;FOLD LIN P2461 Vel=2 m/s CPDAT2461 Tool[1]:marker Base[0] ;%{PE}
;FOLD Parameters ;%{h}
;Params IlfProvider=kukaroboter.basistech.inlineforms.movement.old; Kuka.IsGlobalPoint=False; Kuka.PointName=P2461; Kuka.BlendingEnabled=False; Kuka.MoveDataName=CPDAT1; Kuka.VelocityPath=2; Kuka.CurrentCDSetIndex=0; Kuka.MovementParameterFieldEnabled=True; IlfCommand=LIN
;ENDFOLD
$BWDSTART = FALSE
LDAT_ACT = LCPDAT2461
FDAT_ACT = FP2461
BAS(#CP_PARAMS, 2.0)
SET_CD_PARAMS (0)
LIN XP2461
;ENDFOLD

;FOLD LIN P2462 Vel=2 m/s CPDAT2462 Tool[1]:marker Base[0] ;%{PE}
;FOLD Parameters ;%{h}
;Params IlfProvider=kukaroboter.basistech.inlineforms.movement.old; Kuka.IsGlobalPoint=False; Kuka.PointName=P2462; Kuka.BlendingEnabled=False; Kuka.MoveDataName=CPDAT1; Kuka.VelocityPath=2; Kuka.CurrentCDSetIndex=0; Kuka.MovementParameterFieldEnabled=True; IlfCommand=LIN
;ENDFOLD
$BWDSTART = FALSE
LDAT_ACT = LCPDAT2462
FDAT_ACT = FP2462
BAS(#CP_PARAMS, 2.0)
SET_CD_PARAMS (0)
LIN XP2462
;ENDFOLD

;FOLD LIN P2463 Vel=2 m/s CPDAT2463 Tool[1]:marker Base[0] ;%{PE}
;FOLD Parameters ;%{h}
;Params IlfProvider=kukaroboter.basistech.inlineforms.movement.old; Kuka.IsGlobalPoint=False; Kuka.PointName=P2463; Kuka.BlendingEnabled=False; Kuka.MoveDataName=CPDAT1; Kuka.VelocityPath=2; Kuka.CurrentCDSetIndex=0; Kuka.MovementParameterFieldEnabled=True; IlfCommand=LIN
;ENDFOLD
$BWDSTART = FALSE
LDAT_ACT = LCPDAT2463
FDAT_ACT = FP2463
BAS(#CP_PARAMS, 2.0)
SET_CD_PARAMS (0)
LIN XP2463
;ENDFOLD

;FOLD LIN P2464 Vel=2 m/s CPDAT2464 Tool[1]:marker Base[0] ;%{PE}
;FOLD Parameters ;%{h}
;Params IlfProvider=kukaroboter.basistech.inlineforms.movement.old; Kuka.IsGlobalPoint=False; Kuka.PointName=P2464; Kuka.BlendingEnabled=False; Kuka.MoveDataName=CPDAT1; Kuka.VelocityPath=2; Kuka.CurrentCDSetIndex=0; Kuka.MovementParameterFieldEnabled=True; IlfCommand=LIN
;ENDFOLD
$BWDSTART = FALSE
LDAT_ACT = LCPDAT2464
FDAT_ACT = FP2464
BAS(#CP_PARAMS, 2.0)
SET_CD_PARAMS (0)
LIN XP2464
;ENDFOLD

;FOLD LIN P2465 Vel=2 m/s CPDAT2465 Tool[1]:marker Base[0] ;%{PE}
;FOLD Parameters ;%{h}
;Params IlfProvider=kukaroboter.basistech.inlineforms.movement.old; Kuka.IsGlobalPoint=False; Kuka.PointName=P2465; Kuka.BlendingEnabled=False; Kuka.MoveDataName=CPDAT1; Kuka.VelocityPath=2; Kuka.CurrentCDSetIndex=0; Kuka.MovementParameterFieldEnabled=True; IlfCommand=LIN
;ENDFOLD
$BWDSTART = FALSE
LDAT_ACT = LCPDAT2465
FDAT_ACT = FP2465
BAS(#CP_PARAMS, 2.0)
SET_CD_PARAMS (0)
LIN XP2465
;ENDFOLD

;FOLD LIN P2466 Vel=2 m/s CPDAT2466 Tool[1]:marker Base[0] ;%{PE}
;FOLD Parameters ;%{h}
;Params IlfProvider=kukaroboter.basistech.inlineforms.movement.old; Kuka.IsGlobalPoint=False; Kuka.PointName=P2466; Kuka.BlendingEnabled=False; Kuka.MoveDataName=CPDAT1; Kuka.VelocityPath=2; Kuka.CurrentCDSetIndex=0; Kuka.MovementParameterFieldEnabled=True; IlfCommand=LIN
;ENDFOLD
$BWDSTART = FALSE
LDAT_ACT = LCPDAT2466
FDAT_ACT = FP2466
BAS(#CP_PARAMS, 2.0)
SET_CD_PARAMS (0)
LIN XP2466
;ENDFOLD

;FOLD LIN P2467 Vel=2 m/s CPDAT2467 Tool[1]:marker Base[0] ;%{PE}
;FOLD Parameters ;%{h}
;Params IlfProvider=kukaroboter.basistech.inlineforms.movement.old; Kuka.IsGlobalPoint=False; Kuka.PointName=P2467; Kuka.BlendingEnabled=False; Kuka.MoveDataName=CPDAT1; Kuka.VelocityPath=2; Kuka.CurrentCDSetIndex=0; Kuka.MovementParameterFieldEnabled=True; IlfCommand=LIN
;ENDFOLD
$BWDSTART = FALSE
LDAT_ACT = LCPDAT2467
FDAT_ACT = FP2467
BAS(#CP_PARAMS, 2.0)
SET_CD_PARAMS (0)
LIN XP2467
;ENDFOLD

;FOLD LIN P2468 Vel=2 m/s CPDAT2468 Tool[1]:marker Base[0] ;%{PE}
;FOLD Parameters ;%{h}
;Params IlfProvider=kukaroboter.basistech.inlineforms.movement.old; Kuka.IsGlobalPoint=False; Kuka.PointName=P2468; Kuka.BlendingEnabled=False; Kuka.MoveDataName=CPDAT1; Kuka.VelocityPath=2; Kuka.CurrentCDSetIndex=0; Kuka.MovementParameterFieldEnabled=True; IlfCommand=LIN
;ENDFOLD
$BWDSTART = FALSE
LDAT_ACT = LCPDAT2468
FDAT_ACT = FP2468
BAS(#CP_PARAMS, 2.0)
SET_CD_PARAMS (0)
LIN XP2468
;ENDFOLD

;FOLD LIN P2469 Vel=2 m/s CPDAT2469 Tool[1]:marker Base[0] ;%{PE}
;FOLD Parameters ;%{h}
;Params IlfProvider=kukaroboter.basistech.inlineforms.movement.old; Kuka.IsGlobalPoint=False; Kuka.PointName=P2469; Kuka.BlendingEnabled=False; Kuka.MoveDataName=CPDAT1; Kuka.VelocityPath=2; Kuka.CurrentCDSetIndex=0; Kuka.MovementParameterFieldEnabled=True; IlfCommand=LIN
;ENDFOLD
$BWDSTART = FALSE
LDAT_ACT = LCPDAT2469
FDAT_ACT = FP2469
BAS(#CP_PARAMS, 2.0)
SET_CD_PARAMS (0)
LIN XP2469
;ENDFOLD

;FOLD LIN P2470 Vel=2 m/s CPDAT2470 Tool[1]:marker Base[0] ;%{PE}
;FOLD Parameters ;%{h}
;Params IlfProvider=kukaroboter.basistech.inlineforms.movement.old; Kuka.IsGlobalPoint=False; Kuka.PointName=P2470; Kuka.BlendingEnabled=False; Kuka.MoveDataName=CPDAT1; Kuka.VelocityPath=2; Kuka.CurrentCDSetIndex=0; Kuka.MovementParameterFieldEnabled=True; IlfCommand=LIN
;ENDFOLD
$BWDSTART = FALSE
LDAT_ACT = LCPDAT2470
FDAT_ACT = FP2470
BAS(#CP_PARAMS, 2.0)
SET_CD_PARAMS (0)
LIN XP2470
;ENDFOLD

;FOLD LIN P2471 Vel=2 m/s CPDAT2471 Tool[1]:marker Base[0] ;%{PE}
;FOLD Parameters ;%{h}
;Params IlfProvider=kukaroboter.basistech.inlineforms.movement.old; Kuka.IsGlobalPoint=False; Kuka.PointName=P2471; Kuka.BlendingEnabled=False; Kuka.MoveDataName=CPDAT1; Kuka.VelocityPath=2; Kuka.CurrentCDSetIndex=0; Kuka.MovementParameterFieldEnabled=True; IlfCommand=LIN
;ENDFOLD
$BWDSTART = FALSE
LDAT_ACT = LCPDAT2471
FDAT_ACT = FP2471
BAS(#CP_PARAMS, 2.0)
SET_CD_PARAMS (0)
LIN XP2471
;ENDFOLD

;FOLD LIN P2472 Vel=2 m/s CPDAT2472 Tool[1]:marker Base[0] ;%{PE}
;FOLD Parameters ;%{h}
;Params IlfProvider=kukaroboter.basistech.inlineforms.movement.old; Kuka.IsGlobalPoint=False; Kuka.PointName=P2472; Kuka.BlendingEnabled=False; Kuka.MoveDataName=CPDAT1; Kuka.VelocityPath=2; Kuka.CurrentCDSetIndex=0; Kuka.MovementParameterFieldEnabled=True; IlfCommand=LIN
;ENDFOLD
$BWDSTART = FALSE
LDAT_ACT = LCPDAT2472
FDAT_ACT = FP2472
BAS(#CP_PARAMS, 2.0)
SET_CD_PARAMS (0)
LIN XP2472
;ENDFOLD

;FOLD LIN P2473 Vel=2 m/s CPDAT2473 Tool[1]:marker Base[0] ;%{PE}
;FOLD Parameters ;%{h}
;Params IlfProvider=kukaroboter.basistech.inlineforms.movement.old; Kuka.IsGlobalPoint=False; Kuka.PointName=P2473; Kuka.BlendingEnabled=False; Kuka.MoveDataName=CPDAT1; Kuka.VelocityPath=2; Kuka.CurrentCDSetIndex=0; Kuka.MovementParameterFieldEnabled=True; IlfCommand=LIN
;ENDFOLD
$BWDSTART = FALSE
LDAT_ACT = LCPDAT2473
FDAT_ACT = FP2473
BAS(#CP_PARAMS, 2.0)
SET_CD_PARAMS (0)
LIN XP2473
;ENDFOLD

;FOLD LIN P2474 Vel=2 m/s CPDAT2474 Tool[1]:marker Base[0] ;%{PE}
;FOLD Parameters ;%{h}
;Params IlfProvider=kukaroboter.basistech.inlineforms.movement.old; Kuka.IsGlobalPoint=False; Kuka.PointName=P2474; Kuka.BlendingEnabled=False; Kuka.MoveDataName=CPDAT1; Kuka.VelocityPath=2; Kuka.CurrentCDSetIndex=0; Kuka.MovementParameterFieldEnabled=True; IlfCommand=LIN
;ENDFOLD
$BWDSTART = FALSE
LDAT_ACT = LCPDAT2474
FDAT_ACT = FP2474
BAS(#CP_PARAMS, 2.0)
SET_CD_PARAMS (0)
LIN XP2474
;ENDFOLD

;FOLD LIN P2475 Vel=2 m/s CPDAT2475 Tool[1]:marker Base[0] ;%{PE}
;FOLD Parameters ;%{h}
;Params IlfProvider=kukaroboter.basistech.inlineforms.movement.old; Kuka.IsGlobalPoint=False; Kuka.PointName=P2475; Kuka.BlendingEnabled=False; Kuka.MoveDataName=CPDAT1; Kuka.VelocityPath=2; Kuka.CurrentCDSetIndex=0; Kuka.MovementParameterFieldEnabled=True; IlfCommand=LIN
;ENDFOLD
$BWDSTART = FALSE
LDAT_ACT = LCPDAT2475
FDAT_ACT = FP2475
BAS(#CP_PARAMS, 2.0)
SET_CD_PARAMS (0)
LIN XP2475
;ENDFOLD

;FOLD LIN P2476 Vel=2 m/s CPDAT2476 Tool[1]:marker Base[0] ;%{PE}
;FOLD Parameters ;%{h}
;Params IlfProvider=kukaroboter.basistech.inlineforms.movement.old; Kuka.IsGlobalPoint=False; Kuka.PointName=P2476; Kuka.BlendingEnabled=False; Kuka.MoveDataName=CPDAT1; Kuka.VelocityPath=2; Kuka.CurrentCDSetIndex=0; Kuka.MovementParameterFieldEnabled=True; IlfCommand=LIN
;ENDFOLD
$BWDSTART = FALSE
LDAT_ACT = LCPDAT2476
FDAT_ACT = FP2476
BAS(#CP_PARAMS, 2.0)
SET_CD_PARAMS (0)
LIN XP2476
;ENDFOLD

;FOLD LIN P2477 Vel=2 m/s CPDAT2477 Tool[1]:marker Base[0] ;%{PE}
;FOLD Parameters ;%{h}
;Params IlfProvider=kukaroboter.basistech.inlineforms.movement.old; Kuka.IsGlobalPoint=False; Kuka.PointName=P2477; Kuka.BlendingEnabled=False; Kuka.MoveDataName=CPDAT1; Kuka.VelocityPath=2; Kuka.CurrentCDSetIndex=0; Kuka.MovementParameterFieldEnabled=True; IlfCommand=LIN
;ENDFOLD
$BWDSTART = FALSE
LDAT_ACT = LCPDAT2477
FDAT_ACT = FP2477
BAS(#CP_PARAMS, 2.0)
SET_CD_PARAMS (0)
LIN XP2477
;ENDFOLD

;FOLD LIN P2478 Vel=2 m/s CPDAT2478 Tool[1]:marker Base[0] ;%{PE}
;FOLD Parameters ;%{h}
;Params IlfProvider=kukaroboter.basistech.inlineforms.movement.old; Kuka.IsGlobalPoint=False; Kuka.PointName=P2478; Kuka.BlendingEnabled=False; Kuka.MoveDataName=CPDAT1; Kuka.VelocityPath=2; Kuka.CurrentCDSetIndex=0; Kuka.MovementParameterFieldEnabled=True; IlfCommand=LIN
;ENDFOLD
$BWDSTART = FALSE
LDAT_ACT = LCPDAT2478
FDAT_ACT = FP2478
BAS(#CP_PARAMS, 2.0)
SET_CD_PARAMS (0)
LIN XP2478
;ENDFOLD

;FOLD LIN P2479 Vel=2 m/s CPDAT2479 Tool[1]:marker Base[0] ;%{PE}
;FOLD Parameters ;%{h}
;Params IlfProvider=kukaroboter.basistech.inlineforms.movement.old; Kuka.IsGlobalPoint=False; Kuka.PointName=P2479; Kuka.BlendingEnabled=False; Kuka.MoveDataName=CPDAT1; Kuka.VelocityPath=2; Kuka.CurrentCDSetIndex=0; Kuka.MovementParameterFieldEnabled=True; IlfCommand=LIN
;ENDFOLD
$BWDSTART = FALSE
LDAT_ACT = LCPDAT2479
FDAT_ACT = FP2479
BAS(#CP_PARAMS, 2.0)
SET_CD_PARAMS (0)
LIN XP2479
;ENDFOLD

;FOLD LIN P2480 Vel=2 m/s CPDAT2480 Tool[1]:marker Base[0] ;%{PE}
;FOLD Parameters ;%{h}
;Params IlfProvider=kukaroboter.basistech.inlineforms.movement.old; Kuka.IsGlobalPoint=False; Kuka.PointName=P2480; Kuka.BlendingEnabled=False; Kuka.MoveDataName=CPDAT1; Kuka.VelocityPath=2; Kuka.CurrentCDSetIndex=0; Kuka.MovementParameterFieldEnabled=True; IlfCommand=LIN
;ENDFOLD
$BWDSTART = FALSE
LDAT_ACT = LCPDAT2480
FDAT_ACT = FP2480
BAS(#CP_PARAMS, 2.0)
SET_CD_PARAMS (0)
LIN XP2480
;ENDFOLD

;FOLD LIN P2481 Vel=2 m/s CPDAT2481 Tool[1]:marker Base[0] ;%{PE}
;FOLD Parameters ;%{h}
;Params IlfProvider=kukaroboter.basistech.inlineforms.movement.old; Kuka.IsGlobalPoint=False; Kuka.PointName=P2481; Kuka.BlendingEnabled=False; Kuka.MoveDataName=CPDAT1; Kuka.VelocityPath=2; Kuka.CurrentCDSetIndex=0; Kuka.MovementParameterFieldEnabled=True; IlfCommand=LIN
;ENDFOLD
$BWDSTART = FALSE
LDAT_ACT = LCPDAT2481
FDAT_ACT = FP2481
BAS(#CP_PARAMS, 2.0)
SET_CD_PARAMS (0)
LIN XP2481
;ENDFOLD

;FOLD LIN P2482 Vel=2 m/s CPDAT2482 Tool[1]:marker Base[0] ;%{PE}
;FOLD Parameters ;%{h}
;Params IlfProvider=kukaroboter.basistech.inlineforms.movement.old; Kuka.IsGlobalPoint=False; Kuka.PointName=P2482; Kuka.BlendingEnabled=False; Kuka.MoveDataName=CPDAT1; Kuka.VelocityPath=2; Kuka.CurrentCDSetIndex=0; Kuka.MovementParameterFieldEnabled=True; IlfCommand=LIN
;ENDFOLD
$BWDSTART = FALSE
LDAT_ACT = LCPDAT2482
FDAT_ACT = FP2482
BAS(#CP_PARAMS, 2.0)
SET_CD_PARAMS (0)
LIN XP2482
;ENDFOLD

;FOLD LIN P2483 Vel=2 m/s CPDAT2483 Tool[1]:marker Base[0] ;%{PE}
;FOLD Parameters ;%{h}
;Params IlfProvider=kukaroboter.basistech.inlineforms.movement.old; Kuka.IsGlobalPoint=False; Kuka.PointName=P2483; Kuka.BlendingEnabled=False; Kuka.MoveDataName=CPDAT1; Kuka.VelocityPath=2; Kuka.CurrentCDSetIndex=0; Kuka.MovementParameterFieldEnabled=True; IlfCommand=LIN
;ENDFOLD
$BWDSTART = FALSE
LDAT_ACT = LCPDAT2483
FDAT_ACT = FP2483
BAS(#CP_PARAMS, 2.0)
SET_CD_PARAMS (0)
LIN XP2483
;ENDFOLD

;FOLD LIN P2484 Vel=2 m/s CPDAT2484 Tool[1]:marker Base[0] ;%{PE}
;FOLD Parameters ;%{h}
;Params IlfProvider=kukaroboter.basistech.inlineforms.movement.old; Kuka.IsGlobalPoint=False; Kuka.PointName=P2484; Kuka.BlendingEnabled=False; Kuka.MoveDataName=CPDAT1; Kuka.VelocityPath=2; Kuka.CurrentCDSetIndex=0; Kuka.MovementParameterFieldEnabled=True; IlfCommand=LIN
;ENDFOLD
$BWDSTART = FALSE
LDAT_ACT = LCPDAT2484
FDAT_ACT = FP2484
BAS(#CP_PARAMS, 2.0)
SET_CD_PARAMS (0)
LIN XP2484
;ENDFOLD

;FOLD LIN P2485 Vel=2 m/s CPDAT2485 Tool[1]:marker Base[0] ;%{PE}
;FOLD Parameters ;%{h}
;Params IlfProvider=kukaroboter.basistech.inlineforms.movement.old; Kuka.IsGlobalPoint=False; Kuka.PointName=P2485; Kuka.BlendingEnabled=False; Kuka.MoveDataName=CPDAT1; Kuka.VelocityPath=2; Kuka.CurrentCDSetIndex=0; Kuka.MovementParameterFieldEnabled=True; IlfCommand=LIN
;ENDFOLD
$BWDSTART = FALSE
LDAT_ACT = LCPDAT2485
FDAT_ACT = FP2485
BAS(#CP_PARAMS, 2.0)
SET_CD_PARAMS (0)
LIN XP2485
;ENDFOLD

;FOLD LIN P2486 Vel=2 m/s CPDAT2486 Tool[1]:marker Base[0] ;%{PE}
;FOLD Parameters ;%{h}
;Params IlfProvider=kukaroboter.basistech.inlineforms.movement.old; Kuka.IsGlobalPoint=False; Kuka.PointName=P2486; Kuka.BlendingEnabled=False; Kuka.MoveDataName=CPDAT1; Kuka.VelocityPath=2; Kuka.CurrentCDSetIndex=0; Kuka.MovementParameterFieldEnabled=True; IlfCommand=LIN
;ENDFOLD
$BWDSTART = FALSE
LDAT_ACT = LCPDAT2486
FDAT_ACT = FP2486
BAS(#CP_PARAMS, 2.0)
SET_CD_PARAMS (0)
LIN XP2486
;ENDFOLD

;FOLD LIN P2487 Vel=2 m/s CPDAT2487 Tool[1]:marker Base[0] ;%{PE}
;FOLD Parameters ;%{h}
;Params IlfProvider=kukaroboter.basistech.inlineforms.movement.old; Kuka.IsGlobalPoint=False; Kuka.PointName=P2487; Kuka.BlendingEnabled=False; Kuka.MoveDataName=CPDAT1; Kuka.VelocityPath=2; Kuka.CurrentCDSetIndex=0; Kuka.MovementParameterFieldEnabled=True; IlfCommand=LIN
;ENDFOLD
$BWDSTART = FALSE
LDAT_ACT = LCPDAT2487
FDAT_ACT = FP2487
BAS(#CP_PARAMS, 2.0)
SET_CD_PARAMS (0)
LIN XP2487
;ENDFOLD

;FOLD LIN P2488 Vel=2 m/s CPDAT2488 Tool[1]:marker Base[0] ;%{PE}
;FOLD Parameters ;%{h}
;Params IlfProvider=kukaroboter.basistech.inlineforms.movement.old; Kuka.IsGlobalPoint=False; Kuka.PointName=P2488; Kuka.BlendingEnabled=False; Kuka.MoveDataName=CPDAT1; Kuka.VelocityPath=2; Kuka.CurrentCDSetIndex=0; Kuka.MovementParameterFieldEnabled=True; IlfCommand=LIN
;ENDFOLD
$BWDSTART = FALSE
LDAT_ACT = LCPDAT2488
FDAT_ACT = FP2488
BAS(#CP_PARAMS, 2.0)
SET_CD_PARAMS (0)
LIN XP2488
;ENDFOLD

;FOLD LIN P2489 Vel=2 m/s CPDAT2489 Tool[1]:marker Base[0] ;%{PE}
;FOLD Parameters ;%{h}
;Params IlfProvider=kukaroboter.basistech.inlineforms.movement.old; Kuka.IsGlobalPoint=False; Kuka.PointName=P2489; Kuka.BlendingEnabled=False; Kuka.MoveDataName=CPDAT1; Kuka.VelocityPath=2; Kuka.CurrentCDSetIndex=0; Kuka.MovementParameterFieldEnabled=True; IlfCommand=LIN
;ENDFOLD
$BWDSTART = FALSE
LDAT_ACT = LCPDAT2489
FDAT_ACT = FP2489
BAS(#CP_PARAMS, 2.0)
SET_CD_PARAMS (0)
LIN XP2489
;ENDFOLD

;FOLD LIN P2490 Vel=2 m/s CPDAT2490 Tool[1]:marker Base[0] ;%{PE}
;FOLD Parameters ;%{h}
;Params IlfProvider=kukaroboter.basistech.inlineforms.movement.old; Kuka.IsGlobalPoint=False; Kuka.PointName=P2490; Kuka.BlendingEnabled=False; Kuka.MoveDataName=CPDAT1; Kuka.VelocityPath=2; Kuka.CurrentCDSetIndex=0; Kuka.MovementParameterFieldEnabled=True; IlfCommand=LIN
;ENDFOLD
$BWDSTART = FALSE
LDAT_ACT = LCPDAT2490
FDAT_ACT = FP2490
BAS(#CP_PARAMS, 2.0)
SET_CD_PARAMS (0)
LIN XP2490
;ENDFOLD

;FOLD LIN P2491 Vel=2 m/s CPDAT2491 Tool[1]:marker Base[0] ;%{PE}
;FOLD Parameters ;%{h}
;Params IlfProvider=kukaroboter.basistech.inlineforms.movement.old; Kuka.IsGlobalPoint=False; Kuka.PointName=P2491; Kuka.BlendingEnabled=False; Kuka.MoveDataName=CPDAT1; Kuka.VelocityPath=2; Kuka.CurrentCDSetIndex=0; Kuka.MovementParameterFieldEnabled=True; IlfCommand=LIN
;ENDFOLD
$BWDSTART = FALSE
LDAT_ACT = LCPDAT2491
FDAT_ACT = FP2491
BAS(#CP_PARAMS, 2.0)
SET_CD_PARAMS (0)
LIN XP2491
;ENDFOLD

;FOLD LIN P2492 Vel=2 m/s CPDAT2492 Tool[1]:marker Base[0] ;%{PE}
;FOLD Parameters ;%{h}
;Params IlfProvider=kukaroboter.basistech.inlineforms.movement.old; Kuka.IsGlobalPoint=False; Kuka.PointName=P2492; Kuka.BlendingEnabled=False; Kuka.MoveDataName=CPDAT1; Kuka.VelocityPath=2; Kuka.CurrentCDSetIndex=0; Kuka.MovementParameterFieldEnabled=True; IlfCommand=LIN
;ENDFOLD
$BWDSTART = FALSE
LDAT_ACT = LCPDAT2492
FDAT_ACT = FP2492
BAS(#CP_PARAMS, 2.0)
SET_CD_PARAMS (0)
LIN XP2492
;ENDFOLD

;FOLD LIN P2493 Vel=2 m/s CPDAT2493 Tool[1]:marker Base[0] ;%{PE}
;FOLD Parameters ;%{h}
;Params IlfProvider=kukaroboter.basistech.inlineforms.movement.old; Kuka.IsGlobalPoint=False; Kuka.PointName=P2493; Kuka.BlendingEnabled=False; Kuka.MoveDataName=CPDAT1; Kuka.VelocityPath=2; Kuka.CurrentCDSetIndex=0; Kuka.MovementParameterFieldEnabled=True; IlfCommand=LIN
;ENDFOLD
$BWDSTART = FALSE
LDAT_ACT = LCPDAT2493
FDAT_ACT = FP2493
BAS(#CP_PARAMS, 2.0)
SET_CD_PARAMS (0)
LIN XP2493
;ENDFOLD

;FOLD LIN P2494 Vel=2 m/s CPDAT2494 Tool[1]:marker Base[0] ;%{PE}
;FOLD Parameters ;%{h}
;Params IlfProvider=kukaroboter.basistech.inlineforms.movement.old; Kuka.IsGlobalPoint=False; Kuka.PointName=P2494; Kuka.BlendingEnabled=False; Kuka.MoveDataName=CPDAT1; Kuka.VelocityPath=2; Kuka.CurrentCDSetIndex=0; Kuka.MovementParameterFieldEnabled=True; IlfCommand=LIN
;ENDFOLD
$BWDSTART = FALSE
LDAT_ACT = LCPDAT2494
FDAT_ACT = FP2494
BAS(#CP_PARAMS, 2.0)
SET_CD_PARAMS (0)
LIN XP2494
;ENDFOLD

;FOLD LIN P2495 Vel=2 m/s CPDAT2495 Tool[1]:marker Base[0] ;%{PE}
;FOLD Parameters ;%{h}
;Params IlfProvider=kukaroboter.basistech.inlineforms.movement.old; Kuka.IsGlobalPoint=False; Kuka.PointName=P2495; Kuka.BlendingEnabled=False; Kuka.MoveDataName=CPDAT1; Kuka.VelocityPath=2; Kuka.CurrentCDSetIndex=0; Kuka.MovementParameterFieldEnabled=True; IlfCommand=LIN
;ENDFOLD
$BWDSTART = FALSE
LDAT_ACT = LCPDAT2495
FDAT_ACT = FP2495
BAS(#CP_PARAMS, 2.0)
SET_CD_PARAMS (0)
LIN XP2495
;ENDFOLD

;FOLD LIN P2496 Vel=2 m/s CPDAT2496 Tool[1]:marker Base[0] ;%{PE}
;FOLD Parameters ;%{h}
;Params IlfProvider=kukaroboter.basistech.inlineforms.movement.old; Kuka.IsGlobalPoint=False; Kuka.PointName=P2496; Kuka.BlendingEnabled=False; Kuka.MoveDataName=CPDAT1; Kuka.VelocityPath=2; Kuka.CurrentCDSetIndex=0; Kuka.MovementParameterFieldEnabled=True; IlfCommand=LIN
;ENDFOLD
$BWDSTART = FALSE
LDAT_ACT = LCPDAT2496
FDAT_ACT = FP2496
BAS(#CP_PARAMS, 2.0)
SET_CD_PARAMS (0)
LIN XP2496
;ENDFOLD

;FOLD LIN P2497 Vel=2 m/s CPDAT2497 Tool[1]:marker Base[0] ;%{PE}
;FOLD Parameters ;%{h}
;Params IlfProvider=kukaroboter.basistech.inlineforms.movement.old; Kuka.IsGlobalPoint=False; Kuka.PointName=P2497; Kuka.BlendingEnabled=False; Kuka.MoveDataName=CPDAT1; Kuka.VelocityPath=2; Kuka.CurrentCDSetIndex=0; Kuka.MovementParameterFieldEnabled=True; IlfCommand=LIN
;ENDFOLD
$BWDSTART = FALSE
LDAT_ACT = LCPDAT2497
FDAT_ACT = FP2497
BAS(#CP_PARAMS, 2.0)
SET_CD_PARAMS (0)
LIN XP2497
;ENDFOLD

;FOLD LIN P2498 Vel=2 m/s CPDAT2498 Tool[1]:marker Base[0] ;%{PE}
;FOLD Parameters ;%{h}
;Params IlfProvider=kukaroboter.basistech.inlineforms.movement.old; Kuka.IsGlobalPoint=False; Kuka.PointName=P2498; Kuka.BlendingEnabled=False; Kuka.MoveDataName=CPDAT1; Kuka.VelocityPath=2; Kuka.CurrentCDSetIndex=0; Kuka.MovementParameterFieldEnabled=True; IlfCommand=LIN
;ENDFOLD
$BWDSTART = FALSE
LDAT_ACT = LCPDAT2498
FDAT_ACT = FP2498
BAS(#CP_PARAMS, 2.0)
SET_CD_PARAMS (0)
LIN XP2498
;ENDFOLD

;FOLD LIN P2499 Vel=2 m/s CPDAT2499 Tool[1]:marker Base[0] ;%{PE}
;FOLD Parameters ;%{h}
;Params IlfProvider=kukaroboter.basistech.inlineforms.movement.old; Kuka.IsGlobalPoint=False; Kuka.PointName=P2499; Kuka.BlendingEnabled=False; Kuka.MoveDataName=CPDAT1; Kuka.VelocityPath=2; Kuka.CurrentCDSetIndex=0; Kuka.MovementParameterFieldEnabled=True; IlfCommand=LIN
;ENDFOLD
$BWDSTART = FALSE
LDAT_ACT = LCPDAT2499
FDAT_ACT = FP2499
BAS(#CP_PARAMS, 2.0)
SET_CD_PARAMS (0)
LIN XP2499
;ENDFOLD

;FOLD LIN P2500 Vel=2 m/s CPDAT2500 Tool[1]:marker Base[0] ;%{PE}
;FOLD Parameters ;%{h}
;Params IlfProvider=kukaroboter.basistech.inlineforms.movement.old; Kuka.IsGlobalPoint=False; Kuka.PointName=P2500; Kuka.BlendingEnabled=False; Kuka.MoveDataName=CPDAT1; Kuka.VelocityPath=2; Kuka.CurrentCDSetIndex=0; Kuka.MovementParameterFieldEnabled=True; IlfCommand=LIN
;ENDFOLD
$BWDSTART = FALSE
LDAT_ACT = LCPDAT2500
FDAT_ACT = FP2500
BAS(#CP_PARAMS, 2.0)
SET_CD_PARAMS (0)
LIN XP2500
;ENDFOLD

;FOLD LIN P2501 Vel=2 m/s CPDAT2501 Tool[1]:marker Base[0] ;%{PE}
;FOLD Parameters ;%{h}
;Params IlfProvider=kukaroboter.basistech.inlineforms.movement.old; Kuka.IsGlobalPoint=False; Kuka.PointName=P2501; Kuka.BlendingEnabled=False; Kuka.MoveDataName=CPDAT1; Kuka.VelocityPath=2; Kuka.CurrentCDSetIndex=0; Kuka.MovementParameterFieldEnabled=True; IlfCommand=LIN
;ENDFOLD
$BWDSTART = FALSE
LDAT_ACT = LCPDAT2501
FDAT_ACT = FP2501
BAS(#CP_PARAMS, 2.0)
SET_CD_PARAMS (0)
LIN XP2501
;ENDFOLD

;FOLD LIN P2502 Vel=2 m/s CPDAT2502 Tool[1]:marker Base[0] ;%{PE}
;FOLD Parameters ;%{h}
;Params IlfProvider=kukaroboter.basistech.inlineforms.movement.old; Kuka.IsGlobalPoint=False; Kuka.PointName=P2502; Kuka.BlendingEnabled=False; Kuka.MoveDataName=CPDAT1; Kuka.VelocityPath=2; Kuka.CurrentCDSetIndex=0; Kuka.MovementParameterFieldEnabled=True; IlfCommand=LIN
;ENDFOLD
$BWDSTART = FALSE
LDAT_ACT = LCPDAT2502
FDAT_ACT = FP2502
BAS(#CP_PARAMS, 2.0)
SET_CD_PARAMS (0)
LIN XP2502
;ENDFOLD

;FOLD LIN P2503 Vel=2 m/s CPDAT2503 Tool[1]:marker Base[0] ;%{PE}
;FOLD Parameters ;%{h}
;Params IlfProvider=kukaroboter.basistech.inlineforms.movement.old; Kuka.IsGlobalPoint=False; Kuka.PointName=P2503; Kuka.BlendingEnabled=False; Kuka.MoveDataName=CPDAT1; Kuka.VelocityPath=2; Kuka.CurrentCDSetIndex=0; Kuka.MovementParameterFieldEnabled=True; IlfCommand=LIN
;ENDFOLD
$BWDSTART = FALSE
LDAT_ACT = LCPDAT2503
FDAT_ACT = FP2503
BAS(#CP_PARAMS, 2.0)
SET_CD_PARAMS (0)
LIN XP2503
;ENDFOLD

;FOLD LIN P2504 Vel=2 m/s CPDAT2504 Tool[1]:marker Base[0] ;%{PE}
;FOLD Parameters ;%{h}
;Params IlfProvider=kukaroboter.basistech.inlineforms.movement.old; Kuka.IsGlobalPoint=False; Kuka.PointName=P2504; Kuka.BlendingEnabled=False; Kuka.MoveDataName=CPDAT1; Kuka.VelocityPath=2; Kuka.CurrentCDSetIndex=0; Kuka.MovementParameterFieldEnabled=True; IlfCommand=LIN
;ENDFOLD
$BWDSTART = FALSE
LDAT_ACT = LCPDAT2504
FDAT_ACT = FP2504
BAS(#CP_PARAMS, 2.0)
SET_CD_PARAMS (0)
LIN XP2504
;ENDFOLD

;FOLD LIN P2505 Vel=2 m/s CPDAT2505 Tool[1]:marker Base[0] ;%{PE}
;FOLD Parameters ;%{h}
;Params IlfProvider=kukaroboter.basistech.inlineforms.movement.old; Kuka.IsGlobalPoint=False; Kuka.PointName=P2505; Kuka.BlendingEnabled=False; Kuka.MoveDataName=CPDAT1; Kuka.VelocityPath=2; Kuka.CurrentCDSetIndex=0; Kuka.MovementParameterFieldEnabled=True; IlfCommand=LIN
;ENDFOLD
$BWDSTART = FALSE
LDAT_ACT = LCPDAT2505
FDAT_ACT = FP2505
BAS(#CP_PARAMS, 2.0)
SET_CD_PARAMS (0)
LIN XP2505
;ENDFOLD

;FOLD LIN P2506 Vel=2 m/s CPDAT2506 Tool[1]:marker Base[0] ;%{PE}
;FOLD Parameters ;%{h}
;Params IlfProvider=kukaroboter.basistech.inlineforms.movement.old; Kuka.IsGlobalPoint=False; Kuka.PointName=P2506; Kuka.BlendingEnabled=False; Kuka.MoveDataName=CPDAT1; Kuka.VelocityPath=2; Kuka.CurrentCDSetIndex=0; Kuka.MovementParameterFieldEnabled=True; IlfCommand=LIN
;ENDFOLD
$BWDSTART = FALSE
LDAT_ACT = LCPDAT2506
FDAT_ACT = FP2506
BAS(#CP_PARAMS, 2.0)
SET_CD_PARAMS (0)
LIN XP2506
;ENDFOLD

;FOLD LIN P2507 Vel=2 m/s CPDAT2507 Tool[1]:marker Base[0] ;%{PE}
;FOLD Parameters ;%{h}
;Params IlfProvider=kukaroboter.basistech.inlineforms.movement.old; Kuka.IsGlobalPoint=False; Kuka.PointName=P2507; Kuka.BlendingEnabled=False; Kuka.MoveDataName=CPDAT1; Kuka.VelocityPath=2; Kuka.CurrentCDSetIndex=0; Kuka.MovementParameterFieldEnabled=True; IlfCommand=LIN
;ENDFOLD
$BWDSTART = FALSE
LDAT_ACT = LCPDAT2507
FDAT_ACT = FP2507
BAS(#CP_PARAMS, 2.0)
SET_CD_PARAMS (0)
LIN XP2507
;ENDFOLD

;FOLD LIN P2508 Vel=2 m/s CPDAT2508 Tool[1]:marker Base[0] ;%{PE}
;FOLD Parameters ;%{h}
;Params IlfProvider=kukaroboter.basistech.inlineforms.movement.old; Kuka.IsGlobalPoint=False; Kuka.PointName=P2508; Kuka.BlendingEnabled=False; Kuka.MoveDataName=CPDAT1; Kuka.VelocityPath=2; Kuka.CurrentCDSetIndex=0; Kuka.MovementParameterFieldEnabled=True; IlfCommand=LIN
;ENDFOLD
$BWDSTART = FALSE
LDAT_ACT = LCPDAT2508
FDAT_ACT = FP2508
BAS(#CP_PARAMS, 2.0)
SET_CD_PARAMS (0)
LIN XP2508
;ENDFOLD

;FOLD LIN P2509 Vel=2 m/s CPDAT2509 Tool[1]:marker Base[0] ;%{PE}
;FOLD Parameters ;%{h}
;Params IlfProvider=kukaroboter.basistech.inlineforms.movement.old; Kuka.IsGlobalPoint=False; Kuka.PointName=P2509; Kuka.BlendingEnabled=False; Kuka.MoveDataName=CPDAT1; Kuka.VelocityPath=2; Kuka.CurrentCDSetIndex=0; Kuka.MovementParameterFieldEnabled=True; IlfCommand=LIN
;ENDFOLD
$BWDSTART = FALSE
LDAT_ACT = LCPDAT2509
FDAT_ACT = FP2509
BAS(#CP_PARAMS, 2.0)
SET_CD_PARAMS (0)
LIN XP2509
;ENDFOLD

;FOLD LIN P2510 Vel=2 m/s CPDAT2510 Tool[1]:marker Base[0] ;%{PE}
;FOLD Parameters ;%{h}
;Params IlfProvider=kukaroboter.basistech.inlineforms.movement.old; Kuka.IsGlobalPoint=False; Kuka.PointName=P2510; Kuka.BlendingEnabled=False; Kuka.MoveDataName=CPDAT1; Kuka.VelocityPath=2; Kuka.CurrentCDSetIndex=0; Kuka.MovementParameterFieldEnabled=True; IlfCommand=LIN
;ENDFOLD
$BWDSTART = FALSE
LDAT_ACT = LCPDAT2510
FDAT_ACT = FP2510
BAS(#CP_PARAMS, 2.0)
SET_CD_PARAMS (0)
LIN XP2510
;ENDFOLD

;FOLD LIN P2511 Vel=2 m/s CPDAT2511 Tool[1]:marker Base[0] ;%{PE}
;FOLD Parameters ;%{h}
;Params IlfProvider=kukaroboter.basistech.inlineforms.movement.old; Kuka.IsGlobalPoint=False; Kuka.PointName=P2511; Kuka.BlendingEnabled=False; Kuka.MoveDataName=CPDAT1; Kuka.VelocityPath=2; Kuka.CurrentCDSetIndex=0; Kuka.MovementParameterFieldEnabled=True; IlfCommand=LIN
;ENDFOLD
$BWDSTART = FALSE
LDAT_ACT = LCPDAT2511
FDAT_ACT = FP2511
BAS(#CP_PARAMS, 2.0)
SET_CD_PARAMS (0)
LIN XP2511
;ENDFOLD

;FOLD LIN P2512 Vel=2 m/s CPDAT2512 Tool[1]:marker Base[0] ;%{PE}
;FOLD Parameters ;%{h}
;Params IlfProvider=kukaroboter.basistech.inlineforms.movement.old; Kuka.IsGlobalPoint=False; Kuka.PointName=P2512; Kuka.BlendingEnabled=False; Kuka.MoveDataName=CPDAT1; Kuka.VelocityPath=2; Kuka.CurrentCDSetIndex=0; Kuka.MovementParameterFieldEnabled=True; IlfCommand=LIN
;ENDFOLD
$BWDSTART = FALSE
LDAT_ACT = LCPDAT2512
FDAT_ACT = FP2512
BAS(#CP_PARAMS, 2.0)
SET_CD_PARAMS (0)
LIN XP2512
;ENDFOLD

;FOLD LIN P2513 Vel=2 m/s CPDAT2513 Tool[1]:marker Base[0] ;%{PE}
;FOLD Parameters ;%{h}
;Params IlfProvider=kukaroboter.basistech.inlineforms.movement.old; Kuka.IsGlobalPoint=False; Kuka.PointName=P2513; Kuka.BlendingEnabled=False; Kuka.MoveDataName=CPDAT1; Kuka.VelocityPath=2; Kuka.CurrentCDSetIndex=0; Kuka.MovementParameterFieldEnabled=True; IlfCommand=LIN
;ENDFOLD
$BWDSTART = FALSE
LDAT_ACT = LCPDAT2513
FDAT_ACT = FP2513
BAS(#CP_PARAMS, 2.0)
SET_CD_PARAMS (0)
LIN XP2513
;ENDFOLD

;FOLD LIN P2514 Vel=2 m/s CPDAT2514 Tool[1]:marker Base[0] ;%{PE}
;FOLD Parameters ;%{h}
;Params IlfProvider=kukaroboter.basistech.inlineforms.movement.old; Kuka.IsGlobalPoint=False; Kuka.PointName=P2514; Kuka.BlendingEnabled=False; Kuka.MoveDataName=CPDAT1; Kuka.VelocityPath=2; Kuka.CurrentCDSetIndex=0; Kuka.MovementParameterFieldEnabled=True; IlfCommand=LIN
;ENDFOLD
$BWDSTART = FALSE
LDAT_ACT = LCPDAT2514
FDAT_ACT = FP2514
BAS(#CP_PARAMS, 2.0)
SET_CD_PARAMS (0)
LIN XP2514
;ENDFOLD

;FOLD LIN P2515 Vel=2 m/s CPDAT2515 Tool[1]:marker Base[0] ;%{PE}
;FOLD Parameters ;%{h}
;Params IlfProvider=kukaroboter.basistech.inlineforms.movement.old; Kuka.IsGlobalPoint=False; Kuka.PointName=P2515; Kuka.BlendingEnabled=False; Kuka.MoveDataName=CPDAT1; Kuka.VelocityPath=2; Kuka.CurrentCDSetIndex=0; Kuka.MovementParameterFieldEnabled=True; IlfCommand=LIN
;ENDFOLD
$BWDSTART = FALSE
LDAT_ACT = LCPDAT2515
FDAT_ACT = FP2515
BAS(#CP_PARAMS, 2.0)
SET_CD_PARAMS (0)
LIN XP2515
;ENDFOLD

;FOLD LIN P2516 Vel=2 m/s CPDAT2516 Tool[1]:marker Base[0] ;%{PE}
;FOLD Parameters ;%{h}
;Params IlfProvider=kukaroboter.basistech.inlineforms.movement.old; Kuka.IsGlobalPoint=False; Kuka.PointName=P2516; Kuka.BlendingEnabled=False; Kuka.MoveDataName=CPDAT1; Kuka.VelocityPath=2; Kuka.CurrentCDSetIndex=0; Kuka.MovementParameterFieldEnabled=True; IlfCommand=LIN
;ENDFOLD
$BWDSTART = FALSE
LDAT_ACT = LCPDAT2516
FDAT_ACT = FP2516
BAS(#CP_PARAMS, 2.0)
SET_CD_PARAMS (0)
LIN XP2516
;ENDFOLD

;FOLD LIN P2517 Vel=2 m/s CPDAT2517 Tool[1]:marker Base[0] ;%{PE}
;FOLD Parameters ;%{h}
;Params IlfProvider=kukaroboter.basistech.inlineforms.movement.old; Kuka.IsGlobalPoint=False; Kuka.PointName=P2517; Kuka.BlendingEnabled=False; Kuka.MoveDataName=CPDAT1; Kuka.VelocityPath=2; Kuka.CurrentCDSetIndex=0; Kuka.MovementParameterFieldEnabled=True; IlfCommand=LIN
;ENDFOLD
$BWDSTART = FALSE
LDAT_ACT = LCPDAT2517
FDAT_ACT = FP2517
BAS(#CP_PARAMS, 2.0)
SET_CD_PARAMS (0)
LIN XP2517
;ENDFOLD

;FOLD LIN P2518 Vel=2 m/s CPDAT2518 Tool[1]:marker Base[0] ;%{PE}
;FOLD Parameters ;%{h}
;Params IlfProvider=kukaroboter.basistech.inlineforms.movement.old; Kuka.IsGlobalPoint=False; Kuka.PointName=P2518; Kuka.BlendingEnabled=False; Kuka.MoveDataName=CPDAT1; Kuka.VelocityPath=2; Kuka.CurrentCDSetIndex=0; Kuka.MovementParameterFieldEnabled=True; IlfCommand=LIN
;ENDFOLD
$BWDSTART = FALSE
LDAT_ACT = LCPDAT2518
FDAT_ACT = FP2518
BAS(#CP_PARAMS, 2.0)
SET_CD_PARAMS (0)
LIN XP2518
;ENDFOLD

;FOLD LIN P2519 Vel=2 m/s CPDAT2519 Tool[1]:marker Base[0] ;%{PE}
;FOLD Parameters ;%{h}
;Params IlfProvider=kukaroboter.basistech.inlineforms.movement.old; Kuka.IsGlobalPoint=False; Kuka.PointName=P2519; Kuka.BlendingEnabled=False; Kuka.MoveDataName=CPDAT1; Kuka.VelocityPath=2; Kuka.CurrentCDSetIndex=0; Kuka.MovementParameterFieldEnabled=True; IlfCommand=LIN
;ENDFOLD
$BWDSTART = FALSE
LDAT_ACT = LCPDAT2519
FDAT_ACT = FP2519
BAS(#CP_PARAMS, 2.0)
SET_CD_PARAMS (0)
LIN XP2519
;ENDFOLD

;FOLD LIN P2520 Vel=2 m/s CPDAT2520 Tool[1]:marker Base[0] ;%{PE}
;FOLD Parameters ;%{h}
;Params IlfProvider=kukaroboter.basistech.inlineforms.movement.old; Kuka.IsGlobalPoint=False; Kuka.PointName=P2520; Kuka.BlendingEnabled=False; Kuka.MoveDataName=CPDAT1; Kuka.VelocityPath=2; Kuka.CurrentCDSetIndex=0; Kuka.MovementParameterFieldEnabled=True; IlfCommand=LIN
;ENDFOLD
$BWDSTART = FALSE
LDAT_ACT = LCPDAT2520
FDAT_ACT = FP2520
BAS(#CP_PARAMS, 2.0)
SET_CD_PARAMS (0)
LIN XP2520
;ENDFOLD

;FOLD LIN P2521 Vel=2 m/s CPDAT2521 Tool[1]:marker Base[0] ;%{PE}
;FOLD Parameters ;%{h}
;Params IlfProvider=kukaroboter.basistech.inlineforms.movement.old; Kuka.IsGlobalPoint=False; Kuka.PointName=P2521; Kuka.BlendingEnabled=False; Kuka.MoveDataName=CPDAT1; Kuka.VelocityPath=2; Kuka.CurrentCDSetIndex=0; Kuka.MovementParameterFieldEnabled=True; IlfCommand=LIN
;ENDFOLD
$BWDSTART = FALSE
LDAT_ACT = LCPDAT2521
FDAT_ACT = FP2521
BAS(#CP_PARAMS, 2.0)
SET_CD_PARAMS (0)
LIN XP2521
;ENDFOLD

;FOLD LIN P2522 Vel=2 m/s CPDAT2522 Tool[1]:marker Base[0] ;%{PE}
;FOLD Parameters ;%{h}
;Params IlfProvider=kukaroboter.basistech.inlineforms.movement.old; Kuka.IsGlobalPoint=False; Kuka.PointName=P2522; Kuka.BlendingEnabled=False; Kuka.MoveDataName=CPDAT1; Kuka.VelocityPath=2; Kuka.CurrentCDSetIndex=0; Kuka.MovementParameterFieldEnabled=True; IlfCommand=LIN
;ENDFOLD
$BWDSTART = FALSE
LDAT_ACT = LCPDAT2522
FDAT_ACT = FP2522
BAS(#CP_PARAMS, 2.0)
SET_CD_PARAMS (0)
LIN XP2522
;ENDFOLD

;FOLD LIN P2523 Vel=2 m/s CPDAT2523 Tool[1]:marker Base[0] ;%{PE}
;FOLD Parameters ;%{h}
;Params IlfProvider=kukaroboter.basistech.inlineforms.movement.old; Kuka.IsGlobalPoint=False; Kuka.PointName=P2523; Kuka.BlendingEnabled=False; Kuka.MoveDataName=CPDAT1; Kuka.VelocityPath=2; Kuka.CurrentCDSetIndex=0; Kuka.MovementParameterFieldEnabled=True; IlfCommand=LIN
;ENDFOLD
$BWDSTART = FALSE
LDAT_ACT = LCPDAT2523
FDAT_ACT = FP2523
BAS(#CP_PARAMS, 2.0)
SET_CD_PARAMS (0)
LIN XP2523
;ENDFOLD

;FOLD LIN P2524 Vel=2 m/s CPDAT2524 Tool[1]:marker Base[0] ;%{PE}
;FOLD Parameters ;%{h}
;Params IlfProvider=kukaroboter.basistech.inlineforms.movement.old; Kuka.IsGlobalPoint=False; Kuka.PointName=P2524; Kuka.BlendingEnabled=False; Kuka.MoveDataName=CPDAT1; Kuka.VelocityPath=2; Kuka.CurrentCDSetIndex=0; Kuka.MovementParameterFieldEnabled=True; IlfCommand=LIN
;ENDFOLD
$BWDSTART = FALSE
LDAT_ACT = LCPDAT2524
FDAT_ACT = FP2524
BAS(#CP_PARAMS, 2.0)
SET_CD_PARAMS (0)
LIN XP2524
;ENDFOLD

;FOLD LIN P2525 Vel=2 m/s CPDAT2525 Tool[1]:marker Base[0] ;%{PE}
;FOLD Parameters ;%{h}
;Params IlfProvider=kukaroboter.basistech.inlineforms.movement.old; Kuka.IsGlobalPoint=False; Kuka.PointName=P2525; Kuka.BlendingEnabled=False; Kuka.MoveDataName=CPDAT1; Kuka.VelocityPath=2; Kuka.CurrentCDSetIndex=0; Kuka.MovementParameterFieldEnabled=True; IlfCommand=LIN
;ENDFOLD
$BWDSTART = FALSE
LDAT_ACT = LCPDAT2525
FDAT_ACT = FP2525
BAS(#CP_PARAMS, 2.0)
SET_CD_PARAMS (0)
LIN XP2525
;ENDFOLD

;FOLD LIN P2526 Vel=2 m/s CPDAT2526 Tool[1]:marker Base[0] ;%{PE}
;FOLD Parameters ;%{h}
;Params IlfProvider=kukaroboter.basistech.inlineforms.movement.old; Kuka.IsGlobalPoint=False; Kuka.PointName=P2526; Kuka.BlendingEnabled=False; Kuka.MoveDataName=CPDAT1; Kuka.VelocityPath=2; Kuka.CurrentCDSetIndex=0; Kuka.MovementParameterFieldEnabled=True; IlfCommand=LIN
;ENDFOLD
$BWDSTART = FALSE
LDAT_ACT = LCPDAT2526
FDAT_ACT = FP2526
BAS(#CP_PARAMS, 2.0)
SET_CD_PARAMS (0)
LIN XP2526
;ENDFOLD

;FOLD LIN P2527 Vel=2 m/s CPDAT2527 Tool[1]:marker Base[0] ;%{PE}
;FOLD Parameters ;%{h}
;Params IlfProvider=kukaroboter.basistech.inlineforms.movement.old; Kuka.IsGlobalPoint=False; Kuka.PointName=P2527; Kuka.BlendingEnabled=False; Kuka.MoveDataName=CPDAT1; Kuka.VelocityPath=2; Kuka.CurrentCDSetIndex=0; Kuka.MovementParameterFieldEnabled=True; IlfCommand=LIN
;ENDFOLD
$BWDSTART = FALSE
LDAT_ACT = LCPDAT2527
FDAT_ACT = FP2527
BAS(#CP_PARAMS, 2.0)
SET_CD_PARAMS (0)
LIN XP2527
;ENDFOLD

;FOLD LIN P2528 Vel=2 m/s CPDAT2528 Tool[1]:marker Base[0] ;%{PE}
;FOLD Parameters ;%{h}
;Params IlfProvider=kukaroboter.basistech.inlineforms.movement.old; Kuka.IsGlobalPoint=False; Kuka.PointName=P2528; Kuka.BlendingEnabled=False; Kuka.MoveDataName=CPDAT1; Kuka.VelocityPath=2; Kuka.CurrentCDSetIndex=0; Kuka.MovementParameterFieldEnabled=True; IlfCommand=LIN
;ENDFOLD
$BWDSTART = FALSE
LDAT_ACT = LCPDAT2528
FDAT_ACT = FP2528
BAS(#CP_PARAMS, 2.0)
SET_CD_PARAMS (0)
LIN XP2528
;ENDFOLD

;FOLD LIN P2529 Vel=2 m/s CPDAT2529 Tool[1]:marker Base[0] ;%{PE}
;FOLD Parameters ;%{h}
;Params IlfProvider=kukaroboter.basistech.inlineforms.movement.old; Kuka.IsGlobalPoint=False; Kuka.PointName=P2529; Kuka.BlendingEnabled=False; Kuka.MoveDataName=CPDAT1; Kuka.VelocityPath=2; Kuka.CurrentCDSetIndex=0; Kuka.MovementParameterFieldEnabled=True; IlfCommand=LIN
;ENDFOLD
$BWDSTART = FALSE
LDAT_ACT = LCPDAT2529
FDAT_ACT = FP2529
BAS(#CP_PARAMS, 2.0)
SET_CD_PARAMS (0)
LIN XP2529
;ENDFOLD

;FOLD LIN P2530 Vel=2 m/s CPDAT2530 Tool[1]:marker Base[0] ;%{PE}
;FOLD Parameters ;%{h}
;Params IlfProvider=kukaroboter.basistech.inlineforms.movement.old; Kuka.IsGlobalPoint=False; Kuka.PointName=P2530; Kuka.BlendingEnabled=False; Kuka.MoveDataName=CPDAT1; Kuka.VelocityPath=2; Kuka.CurrentCDSetIndex=0; Kuka.MovementParameterFieldEnabled=True; IlfCommand=LIN
;ENDFOLD
$BWDSTART = FALSE
LDAT_ACT = LCPDAT2530
FDAT_ACT = FP2530
BAS(#CP_PARAMS, 2.0)
SET_CD_PARAMS (0)
LIN XP2530
;ENDFOLD

;FOLD LIN P2531 Vel=2 m/s CPDAT2531 Tool[1]:marker Base[0] ;%{PE}
;FOLD Parameters ;%{h}
;Params IlfProvider=kukaroboter.basistech.inlineforms.movement.old; Kuka.IsGlobalPoint=False; Kuka.PointName=P2531; Kuka.BlendingEnabled=False; Kuka.MoveDataName=CPDAT1; Kuka.VelocityPath=2; Kuka.CurrentCDSetIndex=0; Kuka.MovementParameterFieldEnabled=True; IlfCommand=LIN
;ENDFOLD
$BWDSTART = FALSE
LDAT_ACT = LCPDAT2531
FDAT_ACT = FP2531
BAS(#CP_PARAMS, 2.0)
SET_CD_PARAMS (0)
LIN XP2531
;ENDFOLD

;FOLD LIN P2532 Vel=2 m/s CPDAT2532 Tool[1]:marker Base[0] ;%{PE}
;FOLD Parameters ;%{h}
;Params IlfProvider=kukaroboter.basistech.inlineforms.movement.old; Kuka.IsGlobalPoint=False; Kuka.PointName=P2532; Kuka.BlendingEnabled=False; Kuka.MoveDataName=CPDAT1; Kuka.VelocityPath=2; Kuka.CurrentCDSetIndex=0; Kuka.MovementParameterFieldEnabled=True; IlfCommand=LIN
;ENDFOLD
$BWDSTART = FALSE
LDAT_ACT = LCPDAT2532
FDAT_ACT = FP2532
BAS(#CP_PARAMS, 2.0)
SET_CD_PARAMS (0)
LIN XP2532
;ENDFOLD

;FOLD LIN P2533 Vel=2 m/s CPDAT2533 Tool[1]:marker Base[0] ;%{PE}
;FOLD Parameters ;%{h}
;Params IlfProvider=kukaroboter.basistech.inlineforms.movement.old; Kuka.IsGlobalPoint=False; Kuka.PointName=P2533; Kuka.BlendingEnabled=False; Kuka.MoveDataName=CPDAT1; Kuka.VelocityPath=2; Kuka.CurrentCDSetIndex=0; Kuka.MovementParameterFieldEnabled=True; IlfCommand=LIN
;ENDFOLD
$BWDSTART = FALSE
LDAT_ACT = LCPDAT2533
FDAT_ACT = FP2533
BAS(#CP_PARAMS, 2.0)
SET_CD_PARAMS (0)
LIN XP2533
;ENDFOLD

;FOLD LIN P2534 Vel=2 m/s CPDAT2534 Tool[1]:marker Base[0] ;%{PE}
;FOLD Parameters ;%{h}
;Params IlfProvider=kukaroboter.basistech.inlineforms.movement.old; Kuka.IsGlobalPoint=False; Kuka.PointName=P2534; Kuka.BlendingEnabled=False; Kuka.MoveDataName=CPDAT1; Kuka.VelocityPath=2; Kuka.CurrentCDSetIndex=0; Kuka.MovementParameterFieldEnabled=True; IlfCommand=LIN
;ENDFOLD
$BWDSTART = FALSE
LDAT_ACT = LCPDAT2534
FDAT_ACT = FP2534
BAS(#CP_PARAMS, 2.0)
SET_CD_PARAMS (0)
LIN XP2534
;ENDFOLD

;FOLD LIN P2535 Vel=2 m/s CPDAT2535 Tool[1]:marker Base[0] ;%{PE}
;FOLD Parameters ;%{h}
;Params IlfProvider=kukaroboter.basistech.inlineforms.movement.old; Kuka.IsGlobalPoint=False; Kuka.PointName=P2535; Kuka.BlendingEnabled=False; Kuka.MoveDataName=CPDAT1; Kuka.VelocityPath=2; Kuka.CurrentCDSetIndex=0; Kuka.MovementParameterFieldEnabled=True; IlfCommand=LIN
;ENDFOLD
$BWDSTART = FALSE
LDAT_ACT = LCPDAT2535
FDAT_ACT = FP2535
BAS(#CP_PARAMS, 2.0)
SET_CD_PARAMS (0)
LIN XP2535
;ENDFOLD

;FOLD LIN P2536 Vel=2 m/s CPDAT2536 Tool[1]:marker Base[0] ;%{PE}
;FOLD Parameters ;%{h}
;Params IlfProvider=kukaroboter.basistech.inlineforms.movement.old; Kuka.IsGlobalPoint=False; Kuka.PointName=P2536; Kuka.BlendingEnabled=False; Kuka.MoveDataName=CPDAT1; Kuka.VelocityPath=2; Kuka.CurrentCDSetIndex=0; Kuka.MovementParameterFieldEnabled=True; IlfCommand=LIN
;ENDFOLD
$BWDSTART = FALSE
LDAT_ACT = LCPDAT2536
FDAT_ACT = FP2536
BAS(#CP_PARAMS, 2.0)
SET_CD_PARAMS (0)
LIN XP2536
;ENDFOLD

;FOLD LIN P2537 Vel=2 m/s CPDAT2537 Tool[1]:marker Base[0] ;%{PE}
;FOLD Parameters ;%{h}
;Params IlfProvider=kukaroboter.basistech.inlineforms.movement.old; Kuka.IsGlobalPoint=False; Kuka.PointName=P2537; Kuka.BlendingEnabled=False; Kuka.MoveDataName=CPDAT1; Kuka.VelocityPath=2; Kuka.CurrentCDSetIndex=0; Kuka.MovementParameterFieldEnabled=True; IlfCommand=LIN
;ENDFOLD
$BWDSTART = FALSE
LDAT_ACT = LCPDAT2537
FDAT_ACT = FP2537
BAS(#CP_PARAMS, 2.0)
SET_CD_PARAMS (0)
LIN XP2537
;ENDFOLD

;FOLD LIN P2538 Vel=2 m/s CPDAT2538 Tool[1]:marker Base[0] ;%{PE}
;FOLD Parameters ;%{h}
;Params IlfProvider=kukaroboter.basistech.inlineforms.movement.old; Kuka.IsGlobalPoint=False; Kuka.PointName=P2538; Kuka.BlendingEnabled=False; Kuka.MoveDataName=CPDAT1; Kuka.VelocityPath=2; Kuka.CurrentCDSetIndex=0; Kuka.MovementParameterFieldEnabled=True; IlfCommand=LIN
;ENDFOLD
$BWDSTART = FALSE
LDAT_ACT = LCPDAT2538
FDAT_ACT = FP2538
BAS(#CP_PARAMS, 2.0)
SET_CD_PARAMS (0)
LIN XP2538
;ENDFOLD

;FOLD LIN P2539 Vel=2 m/s CPDAT2539 Tool[1]:marker Base[0] ;%{PE}
;FOLD Parameters ;%{h}
;Params IlfProvider=kukaroboter.basistech.inlineforms.movement.old; Kuka.IsGlobalPoint=False; Kuka.PointName=P2539; Kuka.BlendingEnabled=False; Kuka.MoveDataName=CPDAT1; Kuka.VelocityPath=2; Kuka.CurrentCDSetIndex=0; Kuka.MovementParameterFieldEnabled=True; IlfCommand=LIN
;ENDFOLD
$BWDSTART = FALSE
LDAT_ACT = LCPDAT2539
FDAT_ACT = FP2539
BAS(#CP_PARAMS, 2.0)
SET_CD_PARAMS (0)
LIN XP2539
;ENDFOLD

;FOLD LIN P2540 Vel=2 m/s CPDAT2540 Tool[1]:marker Base[0] ;%{PE}
;FOLD Parameters ;%{h}
;Params IlfProvider=kukaroboter.basistech.inlineforms.movement.old; Kuka.IsGlobalPoint=False; Kuka.PointName=P2540; Kuka.BlendingEnabled=False; Kuka.MoveDataName=CPDAT1; Kuka.VelocityPath=2; Kuka.CurrentCDSetIndex=0; Kuka.MovementParameterFieldEnabled=True; IlfCommand=LIN
;ENDFOLD
$BWDSTART = FALSE
LDAT_ACT = LCPDAT2540
FDAT_ACT = FP2540
BAS(#CP_PARAMS, 2.0)
SET_CD_PARAMS (0)
LIN XP2540
;ENDFOLD

;FOLD LIN P2541 Vel=2 m/s CPDAT2541 Tool[1]:marker Base[0] ;%{PE}
;FOLD Parameters ;%{h}
;Params IlfProvider=kukaroboter.basistech.inlineforms.movement.old; Kuka.IsGlobalPoint=False; Kuka.PointName=P2541; Kuka.BlendingEnabled=False; Kuka.MoveDataName=CPDAT1; Kuka.VelocityPath=2; Kuka.CurrentCDSetIndex=0; Kuka.MovementParameterFieldEnabled=True; IlfCommand=LIN
;ENDFOLD
$BWDSTART = FALSE
LDAT_ACT = LCPDAT2541
FDAT_ACT = FP2541
BAS(#CP_PARAMS, 2.0)
SET_CD_PARAMS (0)
LIN XP2541
;ENDFOLD

;FOLD LIN P2542 Vel=2 m/s CPDAT2542 Tool[1]:marker Base[0] ;%{PE}
;FOLD Parameters ;%{h}
;Params IlfProvider=kukaroboter.basistech.inlineforms.movement.old; Kuka.IsGlobalPoint=False; Kuka.PointName=P2542; Kuka.BlendingEnabled=False; Kuka.MoveDataName=CPDAT1; Kuka.VelocityPath=2; Kuka.CurrentCDSetIndex=0; Kuka.MovementParameterFieldEnabled=True; IlfCommand=LIN
;ENDFOLD
$BWDSTART = FALSE
LDAT_ACT = LCPDAT2542
FDAT_ACT = FP2542
BAS(#CP_PARAMS, 2.0)
SET_CD_PARAMS (0)
LIN XP2542
;ENDFOLD

;FOLD LIN P2543 Vel=2 m/s CPDAT2543 Tool[1]:marker Base[0] ;%{PE}
;FOLD Parameters ;%{h}
;Params IlfProvider=kukaroboter.basistech.inlineforms.movement.old; Kuka.IsGlobalPoint=False; Kuka.PointName=P2543; Kuka.BlendingEnabled=False; Kuka.MoveDataName=CPDAT1; Kuka.VelocityPath=2; Kuka.CurrentCDSetIndex=0; Kuka.MovementParameterFieldEnabled=True; IlfCommand=LIN
;ENDFOLD
$BWDSTART = FALSE
LDAT_ACT = LCPDAT2543
FDAT_ACT = FP2543
BAS(#CP_PARAMS, 2.0)
SET_CD_PARAMS (0)
LIN XP2543
;ENDFOLD

;FOLD LIN P2544 Vel=2 m/s CPDAT2544 Tool[1]:marker Base[0] ;%{PE}
;FOLD Parameters ;%{h}
;Params IlfProvider=kukaroboter.basistech.inlineforms.movement.old; Kuka.IsGlobalPoint=False; Kuka.PointName=P2544; Kuka.BlendingEnabled=False; Kuka.MoveDataName=CPDAT1; Kuka.VelocityPath=2; Kuka.CurrentCDSetIndex=0; Kuka.MovementParameterFieldEnabled=True; IlfCommand=LIN
;ENDFOLD
$BWDSTART = FALSE
LDAT_ACT = LCPDAT2544
FDAT_ACT = FP2544
BAS(#CP_PARAMS, 2.0)
SET_CD_PARAMS (0)
LIN XP2544
;ENDFOLD

;FOLD LIN P2545 Vel=2 m/s CPDAT2545 Tool[1]:marker Base[0] ;%{PE}
;FOLD Parameters ;%{h}
;Params IlfProvider=kukaroboter.basistech.inlineforms.movement.old; Kuka.IsGlobalPoint=False; Kuka.PointName=P2545; Kuka.BlendingEnabled=False; Kuka.MoveDataName=CPDAT1; Kuka.VelocityPath=2; Kuka.CurrentCDSetIndex=0; Kuka.MovementParameterFieldEnabled=True; IlfCommand=LIN
;ENDFOLD
$BWDSTART = FALSE
LDAT_ACT = LCPDAT2545
FDAT_ACT = FP2545
BAS(#CP_PARAMS, 2.0)
SET_CD_PARAMS (0)
LIN XP2545
;ENDFOLD

;FOLD LIN P2546 Vel=2 m/s CPDAT2546 Tool[1]:marker Base[0] ;%{PE}
;FOLD Parameters ;%{h}
;Params IlfProvider=kukaroboter.basistech.inlineforms.movement.old; Kuka.IsGlobalPoint=False; Kuka.PointName=P2546; Kuka.BlendingEnabled=False; Kuka.MoveDataName=CPDAT1; Kuka.VelocityPath=2; Kuka.CurrentCDSetIndex=0; Kuka.MovementParameterFieldEnabled=True; IlfCommand=LIN
;ENDFOLD
$BWDSTART = FALSE
LDAT_ACT = LCPDAT2546
FDAT_ACT = FP2546
BAS(#CP_PARAMS, 2.0)
SET_CD_PARAMS (0)
LIN XP2546
;ENDFOLD

;FOLD LIN P2547 Vel=2 m/s CPDAT2547 Tool[1]:marker Base[0] ;%{PE}
;FOLD Parameters ;%{h}
;Params IlfProvider=kukaroboter.basistech.inlineforms.movement.old; Kuka.IsGlobalPoint=False; Kuka.PointName=P2547; Kuka.BlendingEnabled=False; Kuka.MoveDataName=CPDAT1; Kuka.VelocityPath=2; Kuka.CurrentCDSetIndex=0; Kuka.MovementParameterFieldEnabled=True; IlfCommand=LIN
;ENDFOLD
$BWDSTART = FALSE
LDAT_ACT = LCPDAT2547
FDAT_ACT = FP2547
BAS(#CP_PARAMS, 2.0)
SET_CD_PARAMS (0)
LIN XP2547
;ENDFOLD

;FOLD LIN P2548 Vel=2 m/s CPDAT2548 Tool[1]:marker Base[0] ;%{PE}
;FOLD Parameters ;%{h}
;Params IlfProvider=kukaroboter.basistech.inlineforms.movement.old; Kuka.IsGlobalPoint=False; Kuka.PointName=P2548; Kuka.BlendingEnabled=False; Kuka.MoveDataName=CPDAT1; Kuka.VelocityPath=2; Kuka.CurrentCDSetIndex=0; Kuka.MovementParameterFieldEnabled=True; IlfCommand=LIN
;ENDFOLD
$BWDSTART = FALSE
LDAT_ACT = LCPDAT2548
FDAT_ACT = FP2548
BAS(#CP_PARAMS, 2.0)
SET_CD_PARAMS (0)
LIN XP2548
;ENDFOLD

;FOLD LIN P2549 Vel=2 m/s CPDAT2549 Tool[1]:marker Base[0] ;%{PE}
;FOLD Parameters ;%{h}
;Params IlfProvider=kukaroboter.basistech.inlineforms.movement.old; Kuka.IsGlobalPoint=False; Kuka.PointName=P2549; Kuka.BlendingEnabled=False; Kuka.MoveDataName=CPDAT1; Kuka.VelocityPath=2; Kuka.CurrentCDSetIndex=0; Kuka.MovementParameterFieldEnabled=True; IlfCommand=LIN
;ENDFOLD
$BWDSTART = FALSE
LDAT_ACT = LCPDAT2549
FDAT_ACT = FP2549
BAS(#CP_PARAMS, 2.0)
SET_CD_PARAMS (0)
LIN XP2549
;ENDFOLD

;FOLD LIN P2550 Vel=2 m/s CPDAT2550 Tool[1]:marker Base[0] ;%{PE}
;FOLD Parameters ;%{h}
;Params IlfProvider=kukaroboter.basistech.inlineforms.movement.old; Kuka.IsGlobalPoint=False; Kuka.PointName=P2550; Kuka.BlendingEnabled=False; Kuka.MoveDataName=CPDAT1; Kuka.VelocityPath=2; Kuka.CurrentCDSetIndex=0; Kuka.MovementParameterFieldEnabled=True; IlfCommand=LIN
;ENDFOLD
$BWDSTART = FALSE
LDAT_ACT = LCPDAT2550
FDAT_ACT = FP2550
BAS(#CP_PARAMS, 2.0)
SET_CD_PARAMS (0)
LIN XP2550
;ENDFOLD

;FOLD LIN P2551 Vel=2 m/s CPDAT2551 Tool[1]:marker Base[0] ;%{PE}
;FOLD Parameters ;%{h}
;Params IlfProvider=kukaroboter.basistech.inlineforms.movement.old; Kuka.IsGlobalPoint=False; Kuka.PointName=P2551; Kuka.BlendingEnabled=False; Kuka.MoveDataName=CPDAT1; Kuka.VelocityPath=2; Kuka.CurrentCDSetIndex=0; Kuka.MovementParameterFieldEnabled=True; IlfCommand=LIN
;ENDFOLD
$BWDSTART = FALSE
LDAT_ACT = LCPDAT2551
FDAT_ACT = FP2551
BAS(#CP_PARAMS, 2.0)
SET_CD_PARAMS (0)
LIN XP2551
;ENDFOLD

;FOLD LIN P2552 Vel=2 m/s CPDAT2552 Tool[1]:marker Base[0] ;%{PE}
;FOLD Parameters ;%{h}
;Params IlfProvider=kukaroboter.basistech.inlineforms.movement.old; Kuka.IsGlobalPoint=False; Kuka.PointName=P2552; Kuka.BlendingEnabled=False; Kuka.MoveDataName=CPDAT1; Kuka.VelocityPath=2; Kuka.CurrentCDSetIndex=0; Kuka.MovementParameterFieldEnabled=True; IlfCommand=LIN
;ENDFOLD
$BWDSTART = FALSE
LDAT_ACT = LCPDAT2552
FDAT_ACT = FP2552
BAS(#CP_PARAMS, 2.0)
SET_CD_PARAMS (0)
LIN XP2552
;ENDFOLD

;FOLD LIN P2553 Vel=2 m/s CPDAT2553 Tool[1]:marker Base[0] ;%{PE}
;FOLD Parameters ;%{h}
;Params IlfProvider=kukaroboter.basistech.inlineforms.movement.old; Kuka.IsGlobalPoint=False; Kuka.PointName=P2553; Kuka.BlendingEnabled=False; Kuka.MoveDataName=CPDAT1; Kuka.VelocityPath=2; Kuka.CurrentCDSetIndex=0; Kuka.MovementParameterFieldEnabled=True; IlfCommand=LIN
;ENDFOLD
$BWDSTART = FALSE
LDAT_ACT = LCPDAT2553
FDAT_ACT = FP2553
BAS(#CP_PARAMS, 2.0)
SET_CD_PARAMS (0)
LIN XP2553
;ENDFOLD

;FOLD LIN P2554 Vel=2 m/s CPDAT2554 Tool[1]:marker Base[0] ;%{PE}
;FOLD Parameters ;%{h}
;Params IlfProvider=kukaroboter.basistech.inlineforms.movement.old; Kuka.IsGlobalPoint=False; Kuka.PointName=P2554; Kuka.BlendingEnabled=False; Kuka.MoveDataName=CPDAT1; Kuka.VelocityPath=2; Kuka.CurrentCDSetIndex=0; Kuka.MovementParameterFieldEnabled=True; IlfCommand=LIN
;ENDFOLD
$BWDSTART = FALSE
LDAT_ACT = LCPDAT2554
FDAT_ACT = FP2554
BAS(#CP_PARAMS, 2.0)
SET_CD_PARAMS (0)
LIN XP2554
;ENDFOLD

;FOLD LIN P2555 Vel=2 m/s CPDAT2555 Tool[1]:marker Base[0] ;%{PE}
;FOLD Parameters ;%{h}
;Params IlfProvider=kukaroboter.basistech.inlineforms.movement.old; Kuka.IsGlobalPoint=False; Kuka.PointName=P2555; Kuka.BlendingEnabled=False; Kuka.MoveDataName=CPDAT1; Kuka.VelocityPath=2; Kuka.CurrentCDSetIndex=0; Kuka.MovementParameterFieldEnabled=True; IlfCommand=LIN
;ENDFOLD
$BWDSTART = FALSE
LDAT_ACT = LCPDAT2555
FDAT_ACT = FP2555
BAS(#CP_PARAMS, 2.0)
SET_CD_PARAMS (0)
LIN XP2555
;ENDFOLD

;FOLD LIN P2556 Vel=2 m/s CPDAT2556 Tool[1]:marker Base[0] ;%{PE}
;FOLD Parameters ;%{h}
;Params IlfProvider=kukaroboter.basistech.inlineforms.movement.old; Kuka.IsGlobalPoint=False; Kuka.PointName=P2556; Kuka.BlendingEnabled=False; Kuka.MoveDataName=CPDAT1; Kuka.VelocityPath=2; Kuka.CurrentCDSetIndex=0; Kuka.MovementParameterFieldEnabled=True; IlfCommand=LIN
;ENDFOLD
$BWDSTART = FALSE
LDAT_ACT = LCPDAT2556
FDAT_ACT = FP2556
BAS(#CP_PARAMS, 2.0)
SET_CD_PARAMS (0)
LIN XP2556
;ENDFOLD

;FOLD LIN P2557 Vel=2 m/s CPDAT2557 Tool[1]:marker Base[0] ;%{PE}
;FOLD Parameters ;%{h}
;Params IlfProvider=kukaroboter.basistech.inlineforms.movement.old; Kuka.IsGlobalPoint=False; Kuka.PointName=P2557; Kuka.BlendingEnabled=False; Kuka.MoveDataName=CPDAT1; Kuka.VelocityPath=2; Kuka.CurrentCDSetIndex=0; Kuka.MovementParameterFieldEnabled=True; IlfCommand=LIN
;ENDFOLD
$BWDSTART = FALSE
LDAT_ACT = LCPDAT2557
FDAT_ACT = FP2557
BAS(#CP_PARAMS, 2.0)
SET_CD_PARAMS (0)
LIN XP2557
;ENDFOLD

;FOLD LIN P2558 Vel=2 m/s CPDAT2558 Tool[1]:marker Base[0] ;%{PE}
;FOLD Parameters ;%{h}
;Params IlfProvider=kukaroboter.basistech.inlineforms.movement.old; Kuka.IsGlobalPoint=False; Kuka.PointName=P2558; Kuka.BlendingEnabled=False; Kuka.MoveDataName=CPDAT1; Kuka.VelocityPath=2; Kuka.CurrentCDSetIndex=0; Kuka.MovementParameterFieldEnabled=True; IlfCommand=LIN
;ENDFOLD
$BWDSTART = FALSE
LDAT_ACT = LCPDAT2558
FDAT_ACT = FP2558
BAS(#CP_PARAMS, 2.0)
SET_CD_PARAMS (0)
LIN XP2558
;ENDFOLD

;FOLD LIN P2559 Vel=2 m/s CPDAT2559 Tool[1]:marker Base[0] ;%{PE}
;FOLD Parameters ;%{h}
;Params IlfProvider=kukaroboter.basistech.inlineforms.movement.old; Kuka.IsGlobalPoint=False; Kuka.PointName=P2559; Kuka.BlendingEnabled=False; Kuka.MoveDataName=CPDAT1; Kuka.VelocityPath=2; Kuka.CurrentCDSetIndex=0; Kuka.MovementParameterFieldEnabled=True; IlfCommand=LIN
;ENDFOLD
$BWDSTART = FALSE
LDAT_ACT = LCPDAT2559
FDAT_ACT = FP2559
BAS(#CP_PARAMS, 2.0)
SET_CD_PARAMS (0)
LIN XP2559
;ENDFOLD

;FOLD LIN P2560 Vel=2 m/s CPDAT2560 Tool[1]:marker Base[0] ;%{PE}
;FOLD Parameters ;%{h}
;Params IlfProvider=kukaroboter.basistech.inlineforms.movement.old; Kuka.IsGlobalPoint=False; Kuka.PointName=P2560; Kuka.BlendingEnabled=False; Kuka.MoveDataName=CPDAT1; Kuka.VelocityPath=2; Kuka.CurrentCDSetIndex=0; Kuka.MovementParameterFieldEnabled=True; IlfCommand=LIN
;ENDFOLD
$BWDSTART = FALSE
LDAT_ACT = LCPDAT2560
FDAT_ACT = FP2560
BAS(#CP_PARAMS, 2.0)
SET_CD_PARAMS (0)
LIN XP2560
;ENDFOLD

;FOLD LIN P2561 Vel=2 m/s CPDAT2561 Tool[1]:marker Base[0] ;%{PE}
;FOLD Parameters ;%{h}
;Params IlfProvider=kukaroboter.basistech.inlineforms.movement.old; Kuka.IsGlobalPoint=False; Kuka.PointName=P2561; Kuka.BlendingEnabled=False; Kuka.MoveDataName=CPDAT1; Kuka.VelocityPath=2; Kuka.CurrentCDSetIndex=0; Kuka.MovementParameterFieldEnabled=True; IlfCommand=LIN
;ENDFOLD
$BWDSTART = FALSE
LDAT_ACT = LCPDAT2561
FDAT_ACT = FP2561
BAS(#CP_PARAMS, 2.0)
SET_CD_PARAMS (0)
LIN XP2561
;ENDFOLD

;FOLD LIN P2562 Vel=2 m/s CPDAT2562 Tool[1]:marker Base[0] ;%{PE}
;FOLD Parameters ;%{h}
;Params IlfProvider=kukaroboter.basistech.inlineforms.movement.old; Kuka.IsGlobalPoint=False; Kuka.PointName=P2562; Kuka.BlendingEnabled=False; Kuka.MoveDataName=CPDAT1; Kuka.VelocityPath=2; Kuka.CurrentCDSetIndex=0; Kuka.MovementParameterFieldEnabled=True; IlfCommand=LIN
;ENDFOLD
$BWDSTART = FALSE
LDAT_ACT = LCPDAT2562
FDAT_ACT = FP2562
BAS(#CP_PARAMS, 2.0)
SET_CD_PARAMS (0)
LIN XP2562
;ENDFOLD

;FOLD LIN P2563 Vel=2 m/s CPDAT2563 Tool[1]:marker Base[0] ;%{PE}
;FOLD Parameters ;%{h}
;Params IlfProvider=kukaroboter.basistech.inlineforms.movement.old; Kuka.IsGlobalPoint=False; Kuka.PointName=P2563; Kuka.BlendingEnabled=False; Kuka.MoveDataName=CPDAT1; Kuka.VelocityPath=2; Kuka.CurrentCDSetIndex=0; Kuka.MovementParameterFieldEnabled=True; IlfCommand=LIN
;ENDFOLD
$BWDSTART = FALSE
LDAT_ACT = LCPDAT2563
FDAT_ACT = FP2563
BAS(#CP_PARAMS, 2.0)
SET_CD_PARAMS (0)
LIN XP2563
;ENDFOLD

;FOLD LIN P2564 Vel=2 m/s CPDAT2564 Tool[1]:marker Base[0] ;%{PE}
;FOLD Parameters ;%{h}
;Params IlfProvider=kukaroboter.basistech.inlineforms.movement.old; Kuka.IsGlobalPoint=False; Kuka.PointName=P2564; Kuka.BlendingEnabled=False; Kuka.MoveDataName=CPDAT1; Kuka.VelocityPath=2; Kuka.CurrentCDSetIndex=0; Kuka.MovementParameterFieldEnabled=True; IlfCommand=LIN
;ENDFOLD
$BWDSTART = FALSE
LDAT_ACT = LCPDAT2564
FDAT_ACT = FP2564
BAS(#CP_PARAMS, 2.0)
SET_CD_PARAMS (0)
LIN XP2564
;ENDFOLD

;FOLD LIN P2565 Vel=2 m/s CPDAT2565 Tool[1]:marker Base[0] ;%{PE}
;FOLD Parameters ;%{h}
;Params IlfProvider=kukaroboter.basistech.inlineforms.movement.old; Kuka.IsGlobalPoint=False; Kuka.PointName=P2565; Kuka.BlendingEnabled=False; Kuka.MoveDataName=CPDAT1; Kuka.VelocityPath=2; Kuka.CurrentCDSetIndex=0; Kuka.MovementParameterFieldEnabled=True; IlfCommand=LIN
;ENDFOLD
$BWDSTART = FALSE
LDAT_ACT = LCPDAT2565
FDAT_ACT = FP2565
BAS(#CP_PARAMS, 2.0)
SET_CD_PARAMS (0)
LIN XP2565
;ENDFOLD

;FOLD LIN P2566 Vel=2 m/s CPDAT2566 Tool[1]:marker Base[0] ;%{PE}
;FOLD Parameters ;%{h}
;Params IlfProvider=kukaroboter.basistech.inlineforms.movement.old; Kuka.IsGlobalPoint=False; Kuka.PointName=P2566; Kuka.BlendingEnabled=False; Kuka.MoveDataName=CPDAT1; Kuka.VelocityPath=2; Kuka.CurrentCDSetIndex=0; Kuka.MovementParameterFieldEnabled=True; IlfCommand=LIN
;ENDFOLD
$BWDSTART = FALSE
LDAT_ACT = LCPDAT2566
FDAT_ACT = FP2566
BAS(#CP_PARAMS, 2.0)
SET_CD_PARAMS (0)
LIN XP2566
;ENDFOLD

;FOLD LIN P2567 Vel=2 m/s CPDAT2567 Tool[1]:marker Base[0] ;%{PE}
;FOLD Parameters ;%{h}
;Params IlfProvider=kukaroboter.basistech.inlineforms.movement.old; Kuka.IsGlobalPoint=False; Kuka.PointName=P2567; Kuka.BlendingEnabled=False; Kuka.MoveDataName=CPDAT1; Kuka.VelocityPath=2; Kuka.CurrentCDSetIndex=0; Kuka.MovementParameterFieldEnabled=True; IlfCommand=LIN
;ENDFOLD
$BWDSTART = FALSE
LDAT_ACT = LCPDAT2567
FDAT_ACT = FP2567
BAS(#CP_PARAMS, 2.0)
SET_CD_PARAMS (0)
LIN XP2567
;ENDFOLD

;FOLD LIN P2568 Vel=2 m/s CPDAT2568 Tool[1]:marker Base[0] ;%{PE}
;FOLD Parameters ;%{h}
;Params IlfProvider=kukaroboter.basistech.inlineforms.movement.old; Kuka.IsGlobalPoint=False; Kuka.PointName=P2568; Kuka.BlendingEnabled=False; Kuka.MoveDataName=CPDAT1; Kuka.VelocityPath=2; Kuka.CurrentCDSetIndex=0; Kuka.MovementParameterFieldEnabled=True; IlfCommand=LIN
;ENDFOLD
$BWDSTART = FALSE
LDAT_ACT = LCPDAT2568
FDAT_ACT = FP2568
BAS(#CP_PARAMS, 2.0)
SET_CD_PARAMS (0)
LIN XP2568
;ENDFOLD

;FOLD LIN P2569 Vel=2 m/s CPDAT2569 Tool[1]:marker Base[0] ;%{PE}
;FOLD Parameters ;%{h}
;Params IlfProvider=kukaroboter.basistech.inlineforms.movement.old; Kuka.IsGlobalPoint=False; Kuka.PointName=P2569; Kuka.BlendingEnabled=False; Kuka.MoveDataName=CPDAT1; Kuka.VelocityPath=2; Kuka.CurrentCDSetIndex=0; Kuka.MovementParameterFieldEnabled=True; IlfCommand=LIN
;ENDFOLD
$BWDSTART = FALSE
LDAT_ACT = LCPDAT2569
FDAT_ACT = FP2569
BAS(#CP_PARAMS, 2.0)
SET_CD_PARAMS (0)
LIN XP2569
;ENDFOLD

;FOLD LIN P2570 Vel=2 m/s CPDAT2570 Tool[1]:marker Base[0] ;%{PE}
;FOLD Parameters ;%{h}
;Params IlfProvider=kukaroboter.basistech.inlineforms.movement.old; Kuka.IsGlobalPoint=False; Kuka.PointName=P2570; Kuka.BlendingEnabled=False; Kuka.MoveDataName=CPDAT1; Kuka.VelocityPath=2; Kuka.CurrentCDSetIndex=0; Kuka.MovementParameterFieldEnabled=True; IlfCommand=LIN
;ENDFOLD
$BWDSTART = FALSE
LDAT_ACT = LCPDAT2570
FDAT_ACT = FP2570
BAS(#CP_PARAMS, 2.0)
SET_CD_PARAMS (0)
LIN XP2570
;ENDFOLD

;FOLD LIN P2571 Vel=2 m/s CPDAT2571 Tool[1]:marker Base[0] ;%{PE}
;FOLD Parameters ;%{h}
;Params IlfProvider=kukaroboter.basistech.inlineforms.movement.old; Kuka.IsGlobalPoint=False; Kuka.PointName=P2571; Kuka.BlendingEnabled=False; Kuka.MoveDataName=CPDAT1; Kuka.VelocityPath=2; Kuka.CurrentCDSetIndex=0; Kuka.MovementParameterFieldEnabled=True; IlfCommand=LIN
;ENDFOLD
$BWDSTART = FALSE
LDAT_ACT = LCPDAT2571
FDAT_ACT = FP2571
BAS(#CP_PARAMS, 2.0)
SET_CD_PARAMS (0)
LIN XP2571
;ENDFOLD

;FOLD LIN P2572 Vel=2 m/s CPDAT2572 Tool[1]:marker Base[0] ;%{PE}
;FOLD Parameters ;%{h}
;Params IlfProvider=kukaroboter.basistech.inlineforms.movement.old; Kuka.IsGlobalPoint=False; Kuka.PointName=P2572; Kuka.BlendingEnabled=False; Kuka.MoveDataName=CPDAT1; Kuka.VelocityPath=2; Kuka.CurrentCDSetIndex=0; Kuka.MovementParameterFieldEnabled=True; IlfCommand=LIN
;ENDFOLD
$BWDSTART = FALSE
LDAT_ACT = LCPDAT2572
FDAT_ACT = FP2572
BAS(#CP_PARAMS, 2.0)
SET_CD_PARAMS (0)
LIN XP2572
;ENDFOLD

;FOLD LIN P2573 Vel=2 m/s CPDAT2573 Tool[1]:marker Base[0] ;%{PE}
;FOLD Parameters ;%{h}
;Params IlfProvider=kukaroboter.basistech.inlineforms.movement.old; Kuka.IsGlobalPoint=False; Kuka.PointName=P2573; Kuka.BlendingEnabled=False; Kuka.MoveDataName=CPDAT1; Kuka.VelocityPath=2; Kuka.CurrentCDSetIndex=0; Kuka.MovementParameterFieldEnabled=True; IlfCommand=LIN
;ENDFOLD
$BWDSTART = FALSE
LDAT_ACT = LCPDAT2573
FDAT_ACT = FP2573
BAS(#CP_PARAMS, 2.0)
SET_CD_PARAMS (0)
LIN XP2573
;ENDFOLD

;FOLD LIN P2574 Vel=2 m/s CPDAT2574 Tool[1]:marker Base[0] ;%{PE}
;FOLD Parameters ;%{h}
;Params IlfProvider=kukaroboter.basistech.inlineforms.movement.old; Kuka.IsGlobalPoint=False; Kuka.PointName=P2574; Kuka.BlendingEnabled=False; Kuka.MoveDataName=CPDAT1; Kuka.VelocityPath=2; Kuka.CurrentCDSetIndex=0; Kuka.MovementParameterFieldEnabled=True; IlfCommand=LIN
;ENDFOLD
$BWDSTART = FALSE
LDAT_ACT = LCPDAT2574
FDAT_ACT = FP2574
BAS(#CP_PARAMS, 2.0)
SET_CD_PARAMS (0)
LIN XP2574
;ENDFOLD

;FOLD LIN P2575 Vel=2 m/s CPDAT2575 Tool[1]:marker Base[0] ;%{PE}
;FOLD Parameters ;%{h}
;Params IlfProvider=kukaroboter.basistech.inlineforms.movement.old; Kuka.IsGlobalPoint=False; Kuka.PointName=P2575; Kuka.BlendingEnabled=False; Kuka.MoveDataName=CPDAT1; Kuka.VelocityPath=2; Kuka.CurrentCDSetIndex=0; Kuka.MovementParameterFieldEnabled=True; IlfCommand=LIN
;ENDFOLD
$BWDSTART = FALSE
LDAT_ACT = LCPDAT2575
FDAT_ACT = FP2575
BAS(#CP_PARAMS, 2.0)
SET_CD_PARAMS (0)
LIN XP2575
;ENDFOLD

;FOLD LIN P2576 Vel=2 m/s CPDAT2576 Tool[1]:marker Base[0] ;%{PE}
;FOLD Parameters ;%{h}
;Params IlfProvider=kukaroboter.basistech.inlineforms.movement.old; Kuka.IsGlobalPoint=False; Kuka.PointName=P2576; Kuka.BlendingEnabled=False; Kuka.MoveDataName=CPDAT1; Kuka.VelocityPath=2; Kuka.CurrentCDSetIndex=0; Kuka.MovementParameterFieldEnabled=True; IlfCommand=LIN
;ENDFOLD
$BWDSTART = FALSE
LDAT_ACT = LCPDAT2576
FDAT_ACT = FP2576
BAS(#CP_PARAMS, 2.0)
SET_CD_PARAMS (0)
LIN XP2576
;ENDFOLD

;FOLD LIN P2577 Vel=2 m/s CPDAT2577 Tool[1]:marker Base[0] ;%{PE}
;FOLD Parameters ;%{h}
;Params IlfProvider=kukaroboter.basistech.inlineforms.movement.old; Kuka.IsGlobalPoint=False; Kuka.PointName=P2577; Kuka.BlendingEnabled=False; Kuka.MoveDataName=CPDAT1; Kuka.VelocityPath=2; Kuka.CurrentCDSetIndex=0; Kuka.MovementParameterFieldEnabled=True; IlfCommand=LIN
;ENDFOLD
$BWDSTART = FALSE
LDAT_ACT = LCPDAT2577
FDAT_ACT = FP2577
BAS(#CP_PARAMS, 2.0)
SET_CD_PARAMS (0)
LIN XP2577
;ENDFOLD

;FOLD LIN P2578 Vel=2 m/s CPDAT2578 Tool[1]:marker Base[0] ;%{PE}
;FOLD Parameters ;%{h}
;Params IlfProvider=kukaroboter.basistech.inlineforms.movement.old; Kuka.IsGlobalPoint=False; Kuka.PointName=P2578; Kuka.BlendingEnabled=False; Kuka.MoveDataName=CPDAT1; Kuka.VelocityPath=2; Kuka.CurrentCDSetIndex=0; Kuka.MovementParameterFieldEnabled=True; IlfCommand=LIN
;ENDFOLD
$BWDSTART = FALSE
LDAT_ACT = LCPDAT2578
FDAT_ACT = FP2578
BAS(#CP_PARAMS, 2.0)
SET_CD_PARAMS (0)
LIN XP2578
;ENDFOLD

;FOLD LIN P2579 Vel=2 m/s CPDAT2579 Tool[1]:marker Base[0] ;%{PE}
;FOLD Parameters ;%{h}
;Params IlfProvider=kukaroboter.basistech.inlineforms.movement.old; Kuka.IsGlobalPoint=False; Kuka.PointName=P2579; Kuka.BlendingEnabled=False; Kuka.MoveDataName=CPDAT1; Kuka.VelocityPath=2; Kuka.CurrentCDSetIndex=0; Kuka.MovementParameterFieldEnabled=True; IlfCommand=LIN
;ENDFOLD
$BWDSTART = FALSE
LDAT_ACT = LCPDAT2579
FDAT_ACT = FP2579
BAS(#CP_PARAMS, 2.0)
SET_CD_PARAMS (0)
LIN XP2579
;ENDFOLD

;FOLD LIN P2580 Vel=2 m/s CPDAT2580 Tool[1]:marker Base[0] ;%{PE}
;FOLD Parameters ;%{h}
;Params IlfProvider=kukaroboter.basistech.inlineforms.movement.old; Kuka.IsGlobalPoint=False; Kuka.PointName=P2580; Kuka.BlendingEnabled=False; Kuka.MoveDataName=CPDAT1; Kuka.VelocityPath=2; Kuka.CurrentCDSetIndex=0; Kuka.MovementParameterFieldEnabled=True; IlfCommand=LIN
;ENDFOLD
$BWDSTART = FALSE
LDAT_ACT = LCPDAT2580
FDAT_ACT = FP2580
BAS(#CP_PARAMS, 2.0)
SET_CD_PARAMS (0)
LIN XP2580
;ENDFOLD

;FOLD LIN P2581 Vel=2 m/s CPDAT2581 Tool[1]:marker Base[0] ;%{PE}
;FOLD Parameters ;%{h}
;Params IlfProvider=kukaroboter.basistech.inlineforms.movement.old; Kuka.IsGlobalPoint=False; Kuka.PointName=P2581; Kuka.BlendingEnabled=False; Kuka.MoveDataName=CPDAT1; Kuka.VelocityPath=2; Kuka.CurrentCDSetIndex=0; Kuka.MovementParameterFieldEnabled=True; IlfCommand=LIN
;ENDFOLD
$BWDSTART = FALSE
LDAT_ACT = LCPDAT2581
FDAT_ACT = FP2581
BAS(#CP_PARAMS, 2.0)
SET_CD_PARAMS (0)
LIN XP2581
;ENDFOLD

;FOLD LIN P2582 Vel=2 m/s CPDAT2582 Tool[1]:marker Base[0] ;%{PE}
;FOLD Parameters ;%{h}
;Params IlfProvider=kukaroboter.basistech.inlineforms.movement.old; Kuka.IsGlobalPoint=False; Kuka.PointName=P2582; Kuka.BlendingEnabled=False; Kuka.MoveDataName=CPDAT1; Kuka.VelocityPath=2; Kuka.CurrentCDSetIndex=0; Kuka.MovementParameterFieldEnabled=True; IlfCommand=LIN
;ENDFOLD
$BWDSTART = FALSE
LDAT_ACT = LCPDAT2582
FDAT_ACT = FP2582
BAS(#CP_PARAMS, 2.0)
SET_CD_PARAMS (0)
LIN XP2582
;ENDFOLD

;FOLD LIN P2583 Vel=2 m/s CPDAT2583 Tool[1]:marker Base[0] ;%{PE}
;FOLD Parameters ;%{h}
;Params IlfProvider=kukaroboter.basistech.inlineforms.movement.old; Kuka.IsGlobalPoint=False; Kuka.PointName=P2583; Kuka.BlendingEnabled=False; Kuka.MoveDataName=CPDAT1; Kuka.VelocityPath=2; Kuka.CurrentCDSetIndex=0; Kuka.MovementParameterFieldEnabled=True; IlfCommand=LIN
;ENDFOLD
$BWDSTART = FALSE
LDAT_ACT = LCPDAT2583
FDAT_ACT = FP2583
BAS(#CP_PARAMS, 2.0)
SET_CD_PARAMS (0)
LIN XP2583
;ENDFOLD

;FOLD LIN P2584 Vel=2 m/s CPDAT2584 Tool[1]:marker Base[0] ;%{PE}
;FOLD Parameters ;%{h}
;Params IlfProvider=kukaroboter.basistech.inlineforms.movement.old; Kuka.IsGlobalPoint=False; Kuka.PointName=P2584; Kuka.BlendingEnabled=False; Kuka.MoveDataName=CPDAT1; Kuka.VelocityPath=2; Kuka.CurrentCDSetIndex=0; Kuka.MovementParameterFieldEnabled=True; IlfCommand=LIN
;ENDFOLD
$BWDSTART = FALSE
LDAT_ACT = LCPDAT2584
FDAT_ACT = FP2584
BAS(#CP_PARAMS, 2.0)
SET_CD_PARAMS (0)
LIN XP2584
;ENDFOLD

;FOLD LIN P2585 Vel=2 m/s CPDAT2585 Tool[1]:marker Base[0] ;%{PE}
;FOLD Parameters ;%{h}
;Params IlfProvider=kukaroboter.basistech.inlineforms.movement.old; Kuka.IsGlobalPoint=False; Kuka.PointName=P2585; Kuka.BlendingEnabled=False; Kuka.MoveDataName=CPDAT1; Kuka.VelocityPath=2; Kuka.CurrentCDSetIndex=0; Kuka.MovementParameterFieldEnabled=True; IlfCommand=LIN
;ENDFOLD
$BWDSTART = FALSE
LDAT_ACT = LCPDAT2585
FDAT_ACT = FP2585
BAS(#CP_PARAMS, 2.0)
SET_CD_PARAMS (0)
LIN XP2585
;ENDFOLD

;FOLD LIN P2586 Vel=2 m/s CPDAT2586 Tool[1]:marker Base[0] ;%{PE}
;FOLD Parameters ;%{h}
;Params IlfProvider=kukaroboter.basistech.inlineforms.movement.old; Kuka.IsGlobalPoint=False; Kuka.PointName=P2586; Kuka.BlendingEnabled=False; Kuka.MoveDataName=CPDAT1; Kuka.VelocityPath=2; Kuka.CurrentCDSetIndex=0; Kuka.MovementParameterFieldEnabled=True; IlfCommand=LIN
;ENDFOLD
$BWDSTART = FALSE
LDAT_ACT = LCPDAT2586
FDAT_ACT = FP2586
BAS(#CP_PARAMS, 2.0)
SET_CD_PARAMS (0)
LIN XP2586
;ENDFOLD

;FOLD LIN P2587 Vel=2 m/s CPDAT2587 Tool[1]:marker Base[0] ;%{PE}
;FOLD Parameters ;%{h}
;Params IlfProvider=kukaroboter.basistech.inlineforms.movement.old; Kuka.IsGlobalPoint=False; Kuka.PointName=P2587; Kuka.BlendingEnabled=False; Kuka.MoveDataName=CPDAT1; Kuka.VelocityPath=2; Kuka.CurrentCDSetIndex=0; Kuka.MovementParameterFieldEnabled=True; IlfCommand=LIN
;ENDFOLD
$BWDSTART = FALSE
LDAT_ACT = LCPDAT2587
FDAT_ACT = FP2587
BAS(#CP_PARAMS, 2.0)
SET_CD_PARAMS (0)
LIN XP2587
;ENDFOLD

;FOLD LIN P2588 Vel=2 m/s CPDAT2588 Tool[1]:marker Base[0] ;%{PE}
;FOLD Parameters ;%{h}
;Params IlfProvider=kukaroboter.basistech.inlineforms.movement.old; Kuka.IsGlobalPoint=False; Kuka.PointName=P2588; Kuka.BlendingEnabled=False; Kuka.MoveDataName=CPDAT1; Kuka.VelocityPath=2; Kuka.CurrentCDSetIndex=0; Kuka.MovementParameterFieldEnabled=True; IlfCommand=LIN
;ENDFOLD
$BWDSTART = FALSE
LDAT_ACT = LCPDAT2588
FDAT_ACT = FP2588
BAS(#CP_PARAMS, 2.0)
SET_CD_PARAMS (0)
LIN XP2588
;ENDFOLD

;FOLD LIN P2589 Vel=2 m/s CPDAT2589 Tool[1]:marker Base[0] ;%{PE}
;FOLD Parameters ;%{h}
;Params IlfProvider=kukaroboter.basistech.inlineforms.movement.old; Kuka.IsGlobalPoint=False; Kuka.PointName=P2589; Kuka.BlendingEnabled=False; Kuka.MoveDataName=CPDAT1; Kuka.VelocityPath=2; Kuka.CurrentCDSetIndex=0; Kuka.MovementParameterFieldEnabled=True; IlfCommand=LIN
;ENDFOLD
$BWDSTART = FALSE
LDAT_ACT = LCPDAT2589
FDAT_ACT = FP2589
BAS(#CP_PARAMS, 2.0)
SET_CD_PARAMS (0)
LIN XP2589
;ENDFOLD

;FOLD LIN P2590 Vel=2 m/s CPDAT2590 Tool[1]:marker Base[0] ;%{PE}
;FOLD Parameters ;%{h}
;Params IlfProvider=kukaroboter.basistech.inlineforms.movement.old; Kuka.IsGlobalPoint=False; Kuka.PointName=P2590; Kuka.BlendingEnabled=False; Kuka.MoveDataName=CPDAT1; Kuka.VelocityPath=2; Kuka.CurrentCDSetIndex=0; Kuka.MovementParameterFieldEnabled=True; IlfCommand=LIN
;ENDFOLD
$BWDSTART = FALSE
LDAT_ACT = LCPDAT2590
FDAT_ACT = FP2590
BAS(#CP_PARAMS, 2.0)
SET_CD_PARAMS (0)
LIN XP2590
;ENDFOLD

;FOLD LIN P2591 Vel=2 m/s CPDAT2591 Tool[1]:marker Base[0] ;%{PE}
;FOLD Parameters ;%{h}
;Params IlfProvider=kukaroboter.basistech.inlineforms.movement.old; Kuka.IsGlobalPoint=False; Kuka.PointName=P2591; Kuka.BlendingEnabled=False; Kuka.MoveDataName=CPDAT1; Kuka.VelocityPath=2; Kuka.CurrentCDSetIndex=0; Kuka.MovementParameterFieldEnabled=True; IlfCommand=LIN
;ENDFOLD
$BWDSTART = FALSE
LDAT_ACT = LCPDAT2591
FDAT_ACT = FP2591
BAS(#CP_PARAMS, 2.0)
SET_CD_PARAMS (0)
LIN XP2591
;ENDFOLD

;FOLD LIN P2592 Vel=2 m/s CPDAT2592 Tool[1]:marker Base[0] ;%{PE}
;FOLD Parameters ;%{h}
;Params IlfProvider=kukaroboter.basistech.inlineforms.movement.old; Kuka.IsGlobalPoint=False; Kuka.PointName=P2592; Kuka.BlendingEnabled=False; Kuka.MoveDataName=CPDAT1; Kuka.VelocityPath=2; Kuka.CurrentCDSetIndex=0; Kuka.MovementParameterFieldEnabled=True; IlfCommand=LIN
;ENDFOLD
$BWDSTART = FALSE
LDAT_ACT = LCPDAT2592
FDAT_ACT = FP2592
BAS(#CP_PARAMS, 2.0)
SET_CD_PARAMS (0)
LIN XP2592
;ENDFOLD

;FOLD LIN P2593 Vel=2 m/s CPDAT2593 Tool[1]:marker Base[0] ;%{PE}
;FOLD Parameters ;%{h}
;Params IlfProvider=kukaroboter.basistech.inlineforms.movement.old; Kuka.IsGlobalPoint=False; Kuka.PointName=P2593; Kuka.BlendingEnabled=False; Kuka.MoveDataName=CPDAT1; Kuka.VelocityPath=2; Kuka.CurrentCDSetIndex=0; Kuka.MovementParameterFieldEnabled=True; IlfCommand=LIN
;ENDFOLD
$BWDSTART = FALSE
LDAT_ACT = LCPDAT2593
FDAT_ACT = FP2593
BAS(#CP_PARAMS, 2.0)
SET_CD_PARAMS (0)
LIN XP2593
;ENDFOLD

;FOLD LIN P2594 Vel=2 m/s CPDAT2594 Tool[1]:marker Base[0] ;%{PE}
;FOLD Parameters ;%{h}
;Params IlfProvider=kukaroboter.basistech.inlineforms.movement.old; Kuka.IsGlobalPoint=False; Kuka.PointName=P2594; Kuka.BlendingEnabled=False; Kuka.MoveDataName=CPDAT1; Kuka.VelocityPath=2; Kuka.CurrentCDSetIndex=0; Kuka.MovementParameterFieldEnabled=True; IlfCommand=LIN
;ENDFOLD
$BWDSTART = FALSE
LDAT_ACT = LCPDAT2594
FDAT_ACT = FP2594
BAS(#CP_PARAMS, 2.0)
SET_CD_PARAMS (0)
LIN XP2594
;ENDFOLD

;FOLD LIN P2595 Vel=2 m/s CPDAT2595 Tool[1]:marker Base[0] ;%{PE}
;FOLD Parameters ;%{h}
;Params IlfProvider=kukaroboter.basistech.inlineforms.movement.old; Kuka.IsGlobalPoint=False; Kuka.PointName=P2595; Kuka.BlendingEnabled=False; Kuka.MoveDataName=CPDAT1; Kuka.VelocityPath=2; Kuka.CurrentCDSetIndex=0; Kuka.MovementParameterFieldEnabled=True; IlfCommand=LIN
;ENDFOLD
$BWDSTART = FALSE
LDAT_ACT = LCPDAT2595
FDAT_ACT = FP2595
BAS(#CP_PARAMS, 2.0)
SET_CD_PARAMS (0)
LIN XP2595
;ENDFOLD

;FOLD LIN P2596 Vel=2 m/s CPDAT2596 Tool[1]:marker Base[0] ;%{PE}
;FOLD Parameters ;%{h}
;Params IlfProvider=kukaroboter.basistech.inlineforms.movement.old; Kuka.IsGlobalPoint=False; Kuka.PointName=P2596; Kuka.BlendingEnabled=False; Kuka.MoveDataName=CPDAT1; Kuka.VelocityPath=2; Kuka.CurrentCDSetIndex=0; Kuka.MovementParameterFieldEnabled=True; IlfCommand=LIN
;ENDFOLD
$BWDSTART = FALSE
LDAT_ACT = LCPDAT2596
FDAT_ACT = FP2596
BAS(#CP_PARAMS, 2.0)
SET_CD_PARAMS (0)
LIN XP2596
;ENDFOLD

;FOLD LIN P2597 Vel=2 m/s CPDAT2597 Tool[1]:marker Base[0] ;%{PE}
;FOLD Parameters ;%{h}
;Params IlfProvider=kukaroboter.basistech.inlineforms.movement.old; Kuka.IsGlobalPoint=False; Kuka.PointName=P2597; Kuka.BlendingEnabled=False; Kuka.MoveDataName=CPDAT1; Kuka.VelocityPath=2; Kuka.CurrentCDSetIndex=0; Kuka.MovementParameterFieldEnabled=True; IlfCommand=LIN
;ENDFOLD
$BWDSTART = FALSE
LDAT_ACT = LCPDAT2597
FDAT_ACT = FP2597
BAS(#CP_PARAMS, 2.0)
SET_CD_PARAMS (0)
LIN XP2597
;ENDFOLD

;FOLD LIN P2598 Vel=2 m/s CPDAT2598 Tool[1]:marker Base[0] ;%{PE}
;FOLD Parameters ;%{h}
;Params IlfProvider=kukaroboter.basistech.inlineforms.movement.old; Kuka.IsGlobalPoint=False; Kuka.PointName=P2598; Kuka.BlendingEnabled=False; Kuka.MoveDataName=CPDAT1; Kuka.VelocityPath=2; Kuka.CurrentCDSetIndex=0; Kuka.MovementParameterFieldEnabled=True; IlfCommand=LIN
;ENDFOLD
$BWDSTART = FALSE
LDAT_ACT = LCPDAT2598
FDAT_ACT = FP2598
BAS(#CP_PARAMS, 2.0)
SET_CD_PARAMS (0)
LIN XP2598
;ENDFOLD

;FOLD LIN P2599 Vel=2 m/s CPDAT2599 Tool[1]:marker Base[0] ;%{PE}
;FOLD Parameters ;%{h}
;Params IlfProvider=kukaroboter.basistech.inlineforms.movement.old; Kuka.IsGlobalPoint=False; Kuka.PointName=P2599; Kuka.BlendingEnabled=False; Kuka.MoveDataName=CPDAT1; Kuka.VelocityPath=2; Kuka.CurrentCDSetIndex=0; Kuka.MovementParameterFieldEnabled=True; IlfCommand=LIN
;ENDFOLD
$BWDSTART = FALSE
LDAT_ACT = LCPDAT2599
FDAT_ACT = FP2599
BAS(#CP_PARAMS, 2.0)
SET_CD_PARAMS (0)
LIN XP2599
;ENDFOLD

;FOLD LIN P2600 Vel=2 m/s CPDAT2600 Tool[1]:marker Base[0] ;%{PE}
;FOLD Parameters ;%{h}
;Params IlfProvider=kukaroboter.basistech.inlineforms.movement.old; Kuka.IsGlobalPoint=False; Kuka.PointName=P2600; Kuka.BlendingEnabled=False; Kuka.MoveDataName=CPDAT1; Kuka.VelocityPath=2; Kuka.CurrentCDSetIndex=0; Kuka.MovementParameterFieldEnabled=True; IlfCommand=LIN
;ENDFOLD
$BWDSTART = FALSE
LDAT_ACT = LCPDAT2600
FDAT_ACT = FP2600
BAS(#CP_PARAMS, 2.0)
SET_CD_PARAMS (0)
LIN XP2600
;ENDFOLD

;FOLD LIN P2601 Vel=2 m/s CPDAT2601 Tool[1]:marker Base[0] ;%{PE}
;FOLD Parameters ;%{h}
;Params IlfProvider=kukaroboter.basistech.inlineforms.movement.old; Kuka.IsGlobalPoint=False; Kuka.PointName=P2601; Kuka.BlendingEnabled=False; Kuka.MoveDataName=CPDAT1; Kuka.VelocityPath=2; Kuka.CurrentCDSetIndex=0; Kuka.MovementParameterFieldEnabled=True; IlfCommand=LIN
;ENDFOLD
$BWDSTART = FALSE
LDAT_ACT = LCPDAT2601
FDAT_ACT = FP2601
BAS(#CP_PARAMS, 2.0)
SET_CD_PARAMS (0)
LIN XP2601
;ENDFOLD

;FOLD LIN P2602 Vel=2 m/s CPDAT2602 Tool[1]:marker Base[0] ;%{PE}
;FOLD Parameters ;%{h}
;Params IlfProvider=kukaroboter.basistech.inlineforms.movement.old; Kuka.IsGlobalPoint=False; Kuka.PointName=P2602; Kuka.BlendingEnabled=False; Kuka.MoveDataName=CPDAT1; Kuka.VelocityPath=2; Kuka.CurrentCDSetIndex=0; Kuka.MovementParameterFieldEnabled=True; IlfCommand=LIN
;ENDFOLD
$BWDSTART = FALSE
LDAT_ACT = LCPDAT2602
FDAT_ACT = FP2602
BAS(#CP_PARAMS, 2.0)
SET_CD_PARAMS (0)
LIN XP2602
;ENDFOLD

;FOLD LIN P2603 Vel=2 m/s CPDAT2603 Tool[1]:marker Base[0] ;%{PE}
;FOLD Parameters ;%{h}
;Params IlfProvider=kukaroboter.basistech.inlineforms.movement.old; Kuka.IsGlobalPoint=False; Kuka.PointName=P2603; Kuka.BlendingEnabled=False; Kuka.MoveDataName=CPDAT1; Kuka.VelocityPath=2; Kuka.CurrentCDSetIndex=0; Kuka.MovementParameterFieldEnabled=True; IlfCommand=LIN
;ENDFOLD
$BWDSTART = FALSE
LDAT_ACT = LCPDAT2603
FDAT_ACT = FP2603
BAS(#CP_PARAMS, 2.0)
SET_CD_PARAMS (0)
LIN XP2603
;ENDFOLD

;FOLD LIN P2604 Vel=2 m/s CPDAT2604 Tool[1]:marker Base[0] ;%{PE}
;FOLD Parameters ;%{h}
;Params IlfProvider=kukaroboter.basistech.inlineforms.movement.old; Kuka.IsGlobalPoint=False; Kuka.PointName=P2604; Kuka.BlendingEnabled=False; Kuka.MoveDataName=CPDAT1; Kuka.VelocityPath=2; Kuka.CurrentCDSetIndex=0; Kuka.MovementParameterFieldEnabled=True; IlfCommand=LIN
;ENDFOLD
$BWDSTART = FALSE
LDAT_ACT = LCPDAT2604
FDAT_ACT = FP2604
BAS(#CP_PARAMS, 2.0)
SET_CD_PARAMS (0)
LIN XP2604
;ENDFOLD

;FOLD LIN P2605 Vel=2 m/s CPDAT2605 Tool[1]:marker Base[0] ;%{PE}
;FOLD Parameters ;%{h}
;Params IlfProvider=kukaroboter.basistech.inlineforms.movement.old; Kuka.IsGlobalPoint=False; Kuka.PointName=P2605; Kuka.BlendingEnabled=False; Kuka.MoveDataName=CPDAT1; Kuka.VelocityPath=2; Kuka.CurrentCDSetIndex=0; Kuka.MovementParameterFieldEnabled=True; IlfCommand=LIN
;ENDFOLD
$BWDSTART = FALSE
LDAT_ACT = LCPDAT2605
FDAT_ACT = FP2605
BAS(#CP_PARAMS, 2.0)
SET_CD_PARAMS (0)
LIN XP2605
;ENDFOLD

;FOLD LIN P2606 Vel=2 m/s CPDAT2606 Tool[1]:marker Base[0] ;%{PE}
;FOLD Parameters ;%{h}
;Params IlfProvider=kukaroboter.basistech.inlineforms.movement.old; Kuka.IsGlobalPoint=False; Kuka.PointName=P2606; Kuka.BlendingEnabled=False; Kuka.MoveDataName=CPDAT1; Kuka.VelocityPath=2; Kuka.CurrentCDSetIndex=0; Kuka.MovementParameterFieldEnabled=True; IlfCommand=LIN
;ENDFOLD
$BWDSTART = FALSE
LDAT_ACT = LCPDAT2606
FDAT_ACT = FP2606
BAS(#CP_PARAMS, 2.0)
SET_CD_PARAMS (0)
LIN XP2606
;ENDFOLD

;FOLD LIN P2607 Vel=2 m/s CPDAT2607 Tool[1]:marker Base[0] ;%{PE}
;FOLD Parameters ;%{h}
;Params IlfProvider=kukaroboter.basistech.inlineforms.movement.old; Kuka.IsGlobalPoint=False; Kuka.PointName=P2607; Kuka.BlendingEnabled=False; Kuka.MoveDataName=CPDAT1; Kuka.VelocityPath=2; Kuka.CurrentCDSetIndex=0; Kuka.MovementParameterFieldEnabled=True; IlfCommand=LIN
;ENDFOLD
$BWDSTART = FALSE
LDAT_ACT = LCPDAT2607
FDAT_ACT = FP2607
BAS(#CP_PARAMS, 2.0)
SET_CD_PARAMS (0)
LIN XP2607
;ENDFOLD

;FOLD LIN P2608 Vel=2 m/s CPDAT2608 Tool[1]:marker Base[0] ;%{PE}
;FOLD Parameters ;%{h}
;Params IlfProvider=kukaroboter.basistech.inlineforms.movement.old; Kuka.IsGlobalPoint=False; Kuka.PointName=P2608; Kuka.BlendingEnabled=False; Kuka.MoveDataName=CPDAT1; Kuka.VelocityPath=2; Kuka.CurrentCDSetIndex=0; Kuka.MovementParameterFieldEnabled=True; IlfCommand=LIN
;ENDFOLD
$BWDSTART = FALSE
LDAT_ACT = LCPDAT2608
FDAT_ACT = FP2608
BAS(#CP_PARAMS, 2.0)
SET_CD_PARAMS (0)
LIN XP2608
;ENDFOLD

;FOLD LIN P2609 Vel=2 m/s CPDAT2609 Tool[1]:marker Base[0] ;%{PE}
;FOLD Parameters ;%{h}
;Params IlfProvider=kukaroboter.basistech.inlineforms.movement.old; Kuka.IsGlobalPoint=False; Kuka.PointName=P2609; Kuka.BlendingEnabled=False; Kuka.MoveDataName=CPDAT1; Kuka.VelocityPath=2; Kuka.CurrentCDSetIndex=0; Kuka.MovementParameterFieldEnabled=True; IlfCommand=LIN
;ENDFOLD
$BWDSTART = FALSE
LDAT_ACT = LCPDAT2609
FDAT_ACT = FP2609
BAS(#CP_PARAMS, 2.0)
SET_CD_PARAMS (0)
LIN XP2609
;ENDFOLD

;FOLD LIN P2610 Vel=2 m/s CPDAT2610 Tool[1]:marker Base[0] ;%{PE}
;FOLD Parameters ;%{h}
;Params IlfProvider=kukaroboter.basistech.inlineforms.movement.old; Kuka.IsGlobalPoint=False; Kuka.PointName=P2610; Kuka.BlendingEnabled=False; Kuka.MoveDataName=CPDAT1; Kuka.VelocityPath=2; Kuka.CurrentCDSetIndex=0; Kuka.MovementParameterFieldEnabled=True; IlfCommand=LIN
;ENDFOLD
$BWDSTART = FALSE
LDAT_ACT = LCPDAT2610
FDAT_ACT = FP2610
BAS(#CP_PARAMS, 2.0)
SET_CD_PARAMS (0)
LIN XP2610
;ENDFOLD

;FOLD LIN P2611 Vel=2 m/s CPDAT2611 Tool[1]:marker Base[0] ;%{PE}
;FOLD Parameters ;%{h}
;Params IlfProvider=kukaroboter.basistech.inlineforms.movement.old; Kuka.IsGlobalPoint=False; Kuka.PointName=P2611; Kuka.BlendingEnabled=False; Kuka.MoveDataName=CPDAT1; Kuka.VelocityPath=2; Kuka.CurrentCDSetIndex=0; Kuka.MovementParameterFieldEnabled=True; IlfCommand=LIN
;ENDFOLD
$BWDSTART = FALSE
LDAT_ACT = LCPDAT2611
FDAT_ACT = FP2611
BAS(#CP_PARAMS, 2.0)
SET_CD_PARAMS (0)
LIN XP2611
;ENDFOLD

;FOLD LIN P2612 Vel=2 m/s CPDAT2612 Tool[1]:marker Base[0] ;%{PE}
;FOLD Parameters ;%{h}
;Params IlfProvider=kukaroboter.basistech.inlineforms.movement.old; Kuka.IsGlobalPoint=False; Kuka.PointName=P2612; Kuka.BlendingEnabled=False; Kuka.MoveDataName=CPDAT1; Kuka.VelocityPath=2; Kuka.CurrentCDSetIndex=0; Kuka.MovementParameterFieldEnabled=True; IlfCommand=LIN
;ENDFOLD
$BWDSTART = FALSE
LDAT_ACT = LCPDAT2612
FDAT_ACT = FP2612
BAS(#CP_PARAMS, 2.0)
SET_CD_PARAMS (0)
LIN XP2612
;ENDFOLD

;FOLD LIN P2613 Vel=2 m/s CPDAT2613 Tool[1]:marker Base[0] ;%{PE}
;FOLD Parameters ;%{h}
;Params IlfProvider=kukaroboter.basistech.inlineforms.movement.old; Kuka.IsGlobalPoint=False; Kuka.PointName=P2613; Kuka.BlendingEnabled=False; Kuka.MoveDataName=CPDAT1; Kuka.VelocityPath=2; Kuka.CurrentCDSetIndex=0; Kuka.MovementParameterFieldEnabled=True; IlfCommand=LIN
;ENDFOLD
$BWDSTART = FALSE
LDAT_ACT = LCPDAT2613
FDAT_ACT = FP2613
BAS(#CP_PARAMS, 2.0)
SET_CD_PARAMS (0)
LIN XP2613
;ENDFOLD

;FOLD LIN P2614 Vel=2 m/s CPDAT2614 Tool[1]:marker Base[0] ;%{PE}
;FOLD Parameters ;%{h}
;Params IlfProvider=kukaroboter.basistech.inlineforms.movement.old; Kuka.IsGlobalPoint=False; Kuka.PointName=P2614; Kuka.BlendingEnabled=False; Kuka.MoveDataName=CPDAT1; Kuka.VelocityPath=2; Kuka.CurrentCDSetIndex=0; Kuka.MovementParameterFieldEnabled=True; IlfCommand=LIN
;ENDFOLD
$BWDSTART = FALSE
LDAT_ACT = LCPDAT2614
FDAT_ACT = FP2614
BAS(#CP_PARAMS, 2.0)
SET_CD_PARAMS (0)
LIN XP2614
;ENDFOLD

;FOLD LIN P2615 Vel=2 m/s CPDAT2615 Tool[1]:marker Base[0] ;%{PE}
;FOLD Parameters ;%{h}
;Params IlfProvider=kukaroboter.basistech.inlineforms.movement.old; Kuka.IsGlobalPoint=False; Kuka.PointName=P2615; Kuka.BlendingEnabled=False; Kuka.MoveDataName=CPDAT1; Kuka.VelocityPath=2; Kuka.CurrentCDSetIndex=0; Kuka.MovementParameterFieldEnabled=True; IlfCommand=LIN
;ENDFOLD
$BWDSTART = FALSE
LDAT_ACT = LCPDAT2615
FDAT_ACT = FP2615
BAS(#CP_PARAMS, 2.0)
SET_CD_PARAMS (0)
LIN XP2615
;ENDFOLD

;FOLD LIN P2616 Vel=2 m/s CPDAT2616 Tool[1]:marker Base[0] ;%{PE}
;FOLD Parameters ;%{h}
;Params IlfProvider=kukaroboter.basistech.inlineforms.movement.old; Kuka.IsGlobalPoint=False; Kuka.PointName=P2616; Kuka.BlendingEnabled=False; Kuka.MoveDataName=CPDAT1; Kuka.VelocityPath=2; Kuka.CurrentCDSetIndex=0; Kuka.MovementParameterFieldEnabled=True; IlfCommand=LIN
;ENDFOLD
$BWDSTART = FALSE
LDAT_ACT = LCPDAT2616
FDAT_ACT = FP2616
BAS(#CP_PARAMS, 2.0)
SET_CD_PARAMS (0)
LIN XP2616
;ENDFOLD

;FOLD LIN P2617 Vel=2 m/s CPDAT2617 Tool[1]:marker Base[0] ;%{PE}
;FOLD Parameters ;%{h}
;Params IlfProvider=kukaroboter.basistech.inlineforms.movement.old; Kuka.IsGlobalPoint=False; Kuka.PointName=P2617; Kuka.BlendingEnabled=False; Kuka.MoveDataName=CPDAT1; Kuka.VelocityPath=2; Kuka.CurrentCDSetIndex=0; Kuka.MovementParameterFieldEnabled=True; IlfCommand=LIN
;ENDFOLD
$BWDSTART = FALSE
LDAT_ACT = LCPDAT2617
FDAT_ACT = FP2617
BAS(#CP_PARAMS, 2.0)
SET_CD_PARAMS (0)
LIN XP2617
;ENDFOLD

;FOLD LIN P2618 Vel=2 m/s CPDAT2618 Tool[1]:marker Base[0] ;%{PE}
;FOLD Parameters ;%{h}
;Params IlfProvider=kukaroboter.basistech.inlineforms.movement.old; Kuka.IsGlobalPoint=False; Kuka.PointName=P2618; Kuka.BlendingEnabled=False; Kuka.MoveDataName=CPDAT1; Kuka.VelocityPath=2; Kuka.CurrentCDSetIndex=0; Kuka.MovementParameterFieldEnabled=True; IlfCommand=LIN
;ENDFOLD
$BWDSTART = FALSE
LDAT_ACT = LCPDAT2618
FDAT_ACT = FP2618
BAS(#CP_PARAMS, 2.0)
SET_CD_PARAMS (0)
LIN XP2618
;ENDFOLD

;FOLD LIN P2619 Vel=2 m/s CPDAT2619 Tool[1]:marker Base[0] ;%{PE}
;FOLD Parameters ;%{h}
;Params IlfProvider=kukaroboter.basistech.inlineforms.movement.old; Kuka.IsGlobalPoint=False; Kuka.PointName=P2619; Kuka.BlendingEnabled=False; Kuka.MoveDataName=CPDAT1; Kuka.VelocityPath=2; Kuka.CurrentCDSetIndex=0; Kuka.MovementParameterFieldEnabled=True; IlfCommand=LIN
;ENDFOLD
$BWDSTART = FALSE
LDAT_ACT = LCPDAT2619
FDAT_ACT = FP2619
BAS(#CP_PARAMS, 2.0)
SET_CD_PARAMS (0)
LIN XP2619
;ENDFOLD

;FOLD LIN P2620 Vel=2 m/s CPDAT2620 Tool[1]:marker Base[0] ;%{PE}
;FOLD Parameters ;%{h}
;Params IlfProvider=kukaroboter.basistech.inlineforms.movement.old; Kuka.IsGlobalPoint=False; Kuka.PointName=P2620; Kuka.BlendingEnabled=False; Kuka.MoveDataName=CPDAT1; Kuka.VelocityPath=2; Kuka.CurrentCDSetIndex=0; Kuka.MovementParameterFieldEnabled=True; IlfCommand=LIN
;ENDFOLD
$BWDSTART = FALSE
LDAT_ACT = LCPDAT2620
FDAT_ACT = FP2620
BAS(#CP_PARAMS, 2.0)
SET_CD_PARAMS (0)
LIN XP2620
;ENDFOLD

;FOLD LIN P2621 Vel=2 m/s CPDAT2621 Tool[1]:marker Base[0] ;%{PE}
;FOLD Parameters ;%{h}
;Params IlfProvider=kukaroboter.basistech.inlineforms.movement.old; Kuka.IsGlobalPoint=False; Kuka.PointName=P2621; Kuka.BlendingEnabled=False; Kuka.MoveDataName=CPDAT1; Kuka.VelocityPath=2; Kuka.CurrentCDSetIndex=0; Kuka.MovementParameterFieldEnabled=True; IlfCommand=LIN
;ENDFOLD
$BWDSTART = FALSE
LDAT_ACT = LCPDAT2621
FDAT_ACT = FP2621
BAS(#CP_PARAMS, 2.0)
SET_CD_PARAMS (0)
LIN XP2621
;ENDFOLD

;FOLD LIN P2622 Vel=2 m/s CPDAT2622 Tool[1]:marker Base[0] ;%{PE}
;FOLD Parameters ;%{h}
;Params IlfProvider=kukaroboter.basistech.inlineforms.movement.old; Kuka.IsGlobalPoint=False; Kuka.PointName=P2622; Kuka.BlendingEnabled=False; Kuka.MoveDataName=CPDAT1; Kuka.VelocityPath=2; Kuka.CurrentCDSetIndex=0; Kuka.MovementParameterFieldEnabled=True; IlfCommand=LIN
;ENDFOLD
$BWDSTART = FALSE
LDAT_ACT = LCPDAT2622
FDAT_ACT = FP2622
BAS(#CP_PARAMS, 2.0)
SET_CD_PARAMS (0)
LIN XP2622
;ENDFOLD

;FOLD LIN P2623 Vel=2 m/s CPDAT2623 Tool[1]:marker Base[0] ;%{PE}
;FOLD Parameters ;%{h}
;Params IlfProvider=kukaroboter.basistech.inlineforms.movement.old; Kuka.IsGlobalPoint=False; Kuka.PointName=P2623; Kuka.BlendingEnabled=False; Kuka.MoveDataName=CPDAT1; Kuka.VelocityPath=2; Kuka.CurrentCDSetIndex=0; Kuka.MovementParameterFieldEnabled=True; IlfCommand=LIN
;ENDFOLD
$BWDSTART = FALSE
LDAT_ACT = LCPDAT2623
FDAT_ACT = FP2623
BAS(#CP_PARAMS, 2.0)
SET_CD_PARAMS (0)
LIN XP2623
;ENDFOLD

;FOLD LIN P2624 Vel=2 m/s CPDAT2624 Tool[1]:marker Base[0] ;%{PE}
;FOLD Parameters ;%{h}
;Params IlfProvider=kukaroboter.basistech.inlineforms.movement.old; Kuka.IsGlobalPoint=False; Kuka.PointName=P2624; Kuka.BlendingEnabled=False; Kuka.MoveDataName=CPDAT1; Kuka.VelocityPath=2; Kuka.CurrentCDSetIndex=0; Kuka.MovementParameterFieldEnabled=True; IlfCommand=LIN
;ENDFOLD
$BWDSTART = FALSE
LDAT_ACT = LCPDAT2624
FDAT_ACT = FP2624
BAS(#CP_PARAMS, 2.0)
SET_CD_PARAMS (0)
LIN XP2624
;ENDFOLD

;FOLD LIN P2625 Vel=2 m/s CPDAT2625 Tool[1]:marker Base[0] ;%{PE}
;FOLD Parameters ;%{h}
;Params IlfProvider=kukaroboter.basistech.inlineforms.movement.old; Kuka.IsGlobalPoint=False; Kuka.PointName=P2625; Kuka.BlendingEnabled=False; Kuka.MoveDataName=CPDAT1; Kuka.VelocityPath=2; Kuka.CurrentCDSetIndex=0; Kuka.MovementParameterFieldEnabled=True; IlfCommand=LIN
;ENDFOLD
$BWDSTART = FALSE
LDAT_ACT = LCPDAT2625
FDAT_ACT = FP2625
BAS(#CP_PARAMS, 2.0)
SET_CD_PARAMS (0)
LIN XP2625
;ENDFOLD

;FOLD LIN P2626 Vel=2 m/s CPDAT2626 Tool[1]:marker Base[0] ;%{PE}
;FOLD Parameters ;%{h}
;Params IlfProvider=kukaroboter.basistech.inlineforms.movement.old; Kuka.IsGlobalPoint=False; Kuka.PointName=P2626; Kuka.BlendingEnabled=False; Kuka.MoveDataName=CPDAT1; Kuka.VelocityPath=2; Kuka.CurrentCDSetIndex=0; Kuka.MovementParameterFieldEnabled=True; IlfCommand=LIN
;ENDFOLD
$BWDSTART = FALSE
LDAT_ACT = LCPDAT2626
FDAT_ACT = FP2626
BAS(#CP_PARAMS, 2.0)
SET_CD_PARAMS (0)
LIN XP2626
;ENDFOLD

;FOLD LIN P2627 Vel=2 m/s CPDAT2627 Tool[1]:marker Base[0] ;%{PE}
;FOLD Parameters ;%{h}
;Params IlfProvider=kukaroboter.basistech.inlineforms.movement.old; Kuka.IsGlobalPoint=False; Kuka.PointName=P2627; Kuka.BlendingEnabled=False; Kuka.MoveDataName=CPDAT1; Kuka.VelocityPath=2; Kuka.CurrentCDSetIndex=0; Kuka.MovementParameterFieldEnabled=True; IlfCommand=LIN
;ENDFOLD
$BWDSTART = FALSE
LDAT_ACT = LCPDAT2627
FDAT_ACT = FP2627
BAS(#CP_PARAMS, 2.0)
SET_CD_PARAMS (0)
LIN XP2627
;ENDFOLD

;FOLD LIN P2628 Vel=2 m/s CPDAT2628 Tool[1]:marker Base[0] ;%{PE}
;FOLD Parameters ;%{h}
;Params IlfProvider=kukaroboter.basistech.inlineforms.movement.old; Kuka.IsGlobalPoint=False; Kuka.PointName=P2628; Kuka.BlendingEnabled=False; Kuka.MoveDataName=CPDAT1; Kuka.VelocityPath=2; Kuka.CurrentCDSetIndex=0; Kuka.MovementParameterFieldEnabled=True; IlfCommand=LIN
;ENDFOLD
$BWDSTART = FALSE
LDAT_ACT = LCPDAT2628
FDAT_ACT = FP2628
BAS(#CP_PARAMS, 2.0)
SET_CD_PARAMS (0)
LIN XP2628
;ENDFOLD

;FOLD LIN P2629 Vel=2 m/s CPDAT2629 Tool[1]:marker Base[0] ;%{PE}
;FOLD Parameters ;%{h}
;Params IlfProvider=kukaroboter.basistech.inlineforms.movement.old; Kuka.IsGlobalPoint=False; Kuka.PointName=P2629; Kuka.BlendingEnabled=False; Kuka.MoveDataName=CPDAT1; Kuka.VelocityPath=2; Kuka.CurrentCDSetIndex=0; Kuka.MovementParameterFieldEnabled=True; IlfCommand=LIN
;ENDFOLD
$BWDSTART = FALSE
LDAT_ACT = LCPDAT2629
FDAT_ACT = FP2629
BAS(#CP_PARAMS, 2.0)
SET_CD_PARAMS (0)
LIN XP2629
;ENDFOLD

;FOLD LIN P2630 Vel=2 m/s CPDAT2630 Tool[1]:marker Base[0] ;%{PE}
;FOLD Parameters ;%{h}
;Params IlfProvider=kukaroboter.basistech.inlineforms.movement.old; Kuka.IsGlobalPoint=False; Kuka.PointName=P2630; Kuka.BlendingEnabled=False; Kuka.MoveDataName=CPDAT1; Kuka.VelocityPath=2; Kuka.CurrentCDSetIndex=0; Kuka.MovementParameterFieldEnabled=True; IlfCommand=LIN
;ENDFOLD
$BWDSTART = FALSE
LDAT_ACT = LCPDAT2630
FDAT_ACT = FP2630
BAS(#CP_PARAMS, 2.0)
SET_CD_PARAMS (0)
LIN XP2630
;ENDFOLD

;FOLD LIN P2631 Vel=2 m/s CPDAT2631 Tool[1]:marker Base[0] ;%{PE}
;FOLD Parameters ;%{h}
;Params IlfProvider=kukaroboter.basistech.inlineforms.movement.old; Kuka.IsGlobalPoint=False; Kuka.PointName=P2631; Kuka.BlendingEnabled=False; Kuka.MoveDataName=CPDAT1; Kuka.VelocityPath=2; Kuka.CurrentCDSetIndex=0; Kuka.MovementParameterFieldEnabled=True; IlfCommand=LIN
;ENDFOLD
$BWDSTART = FALSE
LDAT_ACT = LCPDAT2631
FDAT_ACT = FP2631
BAS(#CP_PARAMS, 2.0)
SET_CD_PARAMS (0)
LIN XP2631
;ENDFOLD

;FOLD LIN P2632 Vel=2 m/s CPDAT2632 Tool[1]:marker Base[0] ;%{PE}
;FOLD Parameters ;%{h}
;Params IlfProvider=kukaroboter.basistech.inlineforms.movement.old; Kuka.IsGlobalPoint=False; Kuka.PointName=P2632; Kuka.BlendingEnabled=False; Kuka.MoveDataName=CPDAT1; Kuka.VelocityPath=2; Kuka.CurrentCDSetIndex=0; Kuka.MovementParameterFieldEnabled=True; IlfCommand=LIN
;ENDFOLD
$BWDSTART = FALSE
LDAT_ACT = LCPDAT2632
FDAT_ACT = FP2632
BAS(#CP_PARAMS, 2.0)
SET_CD_PARAMS (0)
LIN XP2632
;ENDFOLD

;FOLD LIN P2633 Vel=2 m/s CPDAT2633 Tool[1]:marker Base[0] ;%{PE}
;FOLD Parameters ;%{h}
;Params IlfProvider=kukaroboter.basistech.inlineforms.movement.old; Kuka.IsGlobalPoint=False; Kuka.PointName=P2633; Kuka.BlendingEnabled=False; Kuka.MoveDataName=CPDAT1; Kuka.VelocityPath=2; Kuka.CurrentCDSetIndex=0; Kuka.MovementParameterFieldEnabled=True; IlfCommand=LIN
;ENDFOLD
$BWDSTART = FALSE
LDAT_ACT = LCPDAT2633
FDAT_ACT = FP2633
BAS(#CP_PARAMS, 2.0)
SET_CD_PARAMS (0)
LIN XP2633
;ENDFOLD

;FOLD LIN P2634 Vel=2 m/s CPDAT2634 Tool[1]:marker Base[0] ;%{PE}
;FOLD Parameters ;%{h}
;Params IlfProvider=kukaroboter.basistech.inlineforms.movement.old; Kuka.IsGlobalPoint=False; Kuka.PointName=P2634; Kuka.BlendingEnabled=False; Kuka.MoveDataName=CPDAT1; Kuka.VelocityPath=2; Kuka.CurrentCDSetIndex=0; Kuka.MovementParameterFieldEnabled=True; IlfCommand=LIN
;ENDFOLD
$BWDSTART = FALSE
LDAT_ACT = LCPDAT2634
FDAT_ACT = FP2634
BAS(#CP_PARAMS, 2.0)
SET_CD_PARAMS (0)
LIN XP2634
;ENDFOLD

;FOLD LIN P2635 Vel=2 m/s CPDAT2635 Tool[1]:marker Base[0] ;%{PE}
;FOLD Parameters ;%{h}
;Params IlfProvider=kukaroboter.basistech.inlineforms.movement.old; Kuka.IsGlobalPoint=False; Kuka.PointName=P2635; Kuka.BlendingEnabled=False; Kuka.MoveDataName=CPDAT1; Kuka.VelocityPath=2; Kuka.CurrentCDSetIndex=0; Kuka.MovementParameterFieldEnabled=True; IlfCommand=LIN
;ENDFOLD
$BWDSTART = FALSE
LDAT_ACT = LCPDAT2635
FDAT_ACT = FP2635
BAS(#CP_PARAMS, 2.0)
SET_CD_PARAMS (0)
LIN XP2635
;ENDFOLD

;FOLD LIN P2636 Vel=2 m/s CPDAT2636 Tool[1]:marker Base[0] ;%{PE}
;FOLD Parameters ;%{h}
;Params IlfProvider=kukaroboter.basistech.inlineforms.movement.old; Kuka.IsGlobalPoint=False; Kuka.PointName=P2636; Kuka.BlendingEnabled=False; Kuka.MoveDataName=CPDAT1; Kuka.VelocityPath=2; Kuka.CurrentCDSetIndex=0; Kuka.MovementParameterFieldEnabled=True; IlfCommand=LIN
;ENDFOLD
$BWDSTART = FALSE
LDAT_ACT = LCPDAT2636
FDAT_ACT = FP2636
BAS(#CP_PARAMS, 2.0)
SET_CD_PARAMS (0)
LIN XP2636
;ENDFOLD

;FOLD LIN P2637 Vel=2 m/s CPDAT2637 Tool[1]:marker Base[0] ;%{PE}
;FOLD Parameters ;%{h}
;Params IlfProvider=kukaroboter.basistech.inlineforms.movement.old; Kuka.IsGlobalPoint=False; Kuka.PointName=P2637; Kuka.BlendingEnabled=False; Kuka.MoveDataName=CPDAT1; Kuka.VelocityPath=2; Kuka.CurrentCDSetIndex=0; Kuka.MovementParameterFieldEnabled=True; IlfCommand=LIN
;ENDFOLD
$BWDSTART = FALSE
LDAT_ACT = LCPDAT2637
FDAT_ACT = FP2637
BAS(#CP_PARAMS, 2.0)
SET_CD_PARAMS (0)
LIN XP2637
;ENDFOLD

;FOLD LIN P2638 Vel=2 m/s CPDAT2638 Tool[1]:marker Base[0] ;%{PE}
;FOLD Parameters ;%{h}
;Params IlfProvider=kukaroboter.basistech.inlineforms.movement.old; Kuka.IsGlobalPoint=False; Kuka.PointName=P2638; Kuka.BlendingEnabled=False; Kuka.MoveDataName=CPDAT1; Kuka.VelocityPath=2; Kuka.CurrentCDSetIndex=0; Kuka.MovementParameterFieldEnabled=True; IlfCommand=LIN
;ENDFOLD
$BWDSTART = FALSE
LDAT_ACT = LCPDAT2638
FDAT_ACT = FP2638
BAS(#CP_PARAMS, 2.0)
SET_CD_PARAMS (0)
LIN XP2638
;ENDFOLD

;FOLD LIN P2639 Vel=2 m/s CPDAT2639 Tool[1]:marker Base[0] ;%{PE}
;FOLD Parameters ;%{h}
;Params IlfProvider=kukaroboter.basistech.inlineforms.movement.old; Kuka.IsGlobalPoint=False; Kuka.PointName=P2639; Kuka.BlendingEnabled=False; Kuka.MoveDataName=CPDAT1; Kuka.VelocityPath=2; Kuka.CurrentCDSetIndex=0; Kuka.MovementParameterFieldEnabled=True; IlfCommand=LIN
;ENDFOLD
$BWDSTART = FALSE
LDAT_ACT = LCPDAT2639
FDAT_ACT = FP2639
BAS(#CP_PARAMS, 2.0)
SET_CD_PARAMS (0)
LIN XP2639
;ENDFOLD

;FOLD LIN P2640 Vel=2 m/s CPDAT2640 Tool[1]:marker Base[0] ;%{PE}
;FOLD Parameters ;%{h}
;Params IlfProvider=kukaroboter.basistech.inlineforms.movement.old; Kuka.IsGlobalPoint=False; Kuka.PointName=P2640; Kuka.BlendingEnabled=False; Kuka.MoveDataName=CPDAT1; Kuka.VelocityPath=2; Kuka.CurrentCDSetIndex=0; Kuka.MovementParameterFieldEnabled=True; IlfCommand=LIN
;ENDFOLD
$BWDSTART = FALSE
LDAT_ACT = LCPDAT2640
FDAT_ACT = FP2640
BAS(#CP_PARAMS, 2.0)
SET_CD_PARAMS (0)
LIN XP2640
;ENDFOLD

;FOLD LIN P2641 Vel=2 m/s CPDAT2641 Tool[1]:marker Base[0] ;%{PE}
;FOLD Parameters ;%{h}
;Params IlfProvider=kukaroboter.basistech.inlineforms.movement.old; Kuka.IsGlobalPoint=False; Kuka.PointName=P2641; Kuka.BlendingEnabled=False; Kuka.MoveDataName=CPDAT1; Kuka.VelocityPath=2; Kuka.CurrentCDSetIndex=0; Kuka.MovementParameterFieldEnabled=True; IlfCommand=LIN
;ENDFOLD
$BWDSTART = FALSE
LDAT_ACT = LCPDAT2641
FDAT_ACT = FP2641
BAS(#CP_PARAMS, 2.0)
SET_CD_PARAMS (0)
LIN XP2641
;ENDFOLD

;FOLD LIN P2642 Vel=2 m/s CPDAT2642 Tool[1]:marker Base[0] ;%{PE}
;FOLD Parameters ;%{h}
;Params IlfProvider=kukaroboter.basistech.inlineforms.movement.old; Kuka.IsGlobalPoint=False; Kuka.PointName=P2642; Kuka.BlendingEnabled=False; Kuka.MoveDataName=CPDAT1; Kuka.VelocityPath=2; Kuka.CurrentCDSetIndex=0; Kuka.MovementParameterFieldEnabled=True; IlfCommand=LIN
;ENDFOLD
$BWDSTART = FALSE
LDAT_ACT = LCPDAT2642
FDAT_ACT = FP2642
BAS(#CP_PARAMS, 2.0)
SET_CD_PARAMS (0)
LIN XP2642
;ENDFOLD

;FOLD LIN P2643 Vel=2 m/s CPDAT2643 Tool[1]:marker Base[0] ;%{PE}
;FOLD Parameters ;%{h}
;Params IlfProvider=kukaroboter.basistech.inlineforms.movement.old; Kuka.IsGlobalPoint=False; Kuka.PointName=P2643; Kuka.BlendingEnabled=False; Kuka.MoveDataName=CPDAT1; Kuka.VelocityPath=2; Kuka.CurrentCDSetIndex=0; Kuka.MovementParameterFieldEnabled=True; IlfCommand=LIN
;ENDFOLD
$BWDSTART = FALSE
LDAT_ACT = LCPDAT2643
FDAT_ACT = FP2643
BAS(#CP_PARAMS, 2.0)
SET_CD_PARAMS (0)
LIN XP2643
;ENDFOLD

;FOLD LIN P2644 Vel=2 m/s CPDAT2644 Tool[1]:marker Base[0] ;%{PE}
;FOLD Parameters ;%{h}
;Params IlfProvider=kukaroboter.basistech.inlineforms.movement.old; Kuka.IsGlobalPoint=False; Kuka.PointName=P2644; Kuka.BlendingEnabled=False; Kuka.MoveDataName=CPDAT1; Kuka.VelocityPath=2; Kuka.CurrentCDSetIndex=0; Kuka.MovementParameterFieldEnabled=True; IlfCommand=LIN
;ENDFOLD
$BWDSTART = FALSE
LDAT_ACT = LCPDAT2644
FDAT_ACT = FP2644
BAS(#CP_PARAMS, 2.0)
SET_CD_PARAMS (0)
LIN XP2644
;ENDFOLD

;FOLD LIN P2645 Vel=2 m/s CPDAT2645 Tool[1]:marker Base[0] ;%{PE}
;FOLD Parameters ;%{h}
;Params IlfProvider=kukaroboter.basistech.inlineforms.movement.old; Kuka.IsGlobalPoint=False; Kuka.PointName=P2645; Kuka.BlendingEnabled=False; Kuka.MoveDataName=CPDAT1; Kuka.VelocityPath=2; Kuka.CurrentCDSetIndex=0; Kuka.MovementParameterFieldEnabled=True; IlfCommand=LIN
;ENDFOLD
$BWDSTART = FALSE
LDAT_ACT = LCPDAT2645
FDAT_ACT = FP2645
BAS(#CP_PARAMS, 2.0)
SET_CD_PARAMS (0)
LIN XP2645
;ENDFOLD

;FOLD LIN P2646 Vel=2 m/s CPDAT2646 Tool[1]:marker Base[0] ;%{PE}
;FOLD Parameters ;%{h}
;Params IlfProvider=kukaroboter.basistech.inlineforms.movement.old; Kuka.IsGlobalPoint=False; Kuka.PointName=P2646; Kuka.BlendingEnabled=False; Kuka.MoveDataName=CPDAT1; Kuka.VelocityPath=2; Kuka.CurrentCDSetIndex=0; Kuka.MovementParameterFieldEnabled=True; IlfCommand=LIN
;ENDFOLD
$BWDSTART = FALSE
LDAT_ACT = LCPDAT2646
FDAT_ACT = FP2646
BAS(#CP_PARAMS, 2.0)
SET_CD_PARAMS (0)
LIN XP2646
;ENDFOLD

;FOLD LIN P2647 Vel=2 m/s CPDAT2647 Tool[1]:marker Base[0] ;%{PE}
;FOLD Parameters ;%{h}
;Params IlfProvider=kukaroboter.basistech.inlineforms.movement.old; Kuka.IsGlobalPoint=False; Kuka.PointName=P2647; Kuka.BlendingEnabled=False; Kuka.MoveDataName=CPDAT1; Kuka.VelocityPath=2; Kuka.CurrentCDSetIndex=0; Kuka.MovementParameterFieldEnabled=True; IlfCommand=LIN
;ENDFOLD
$BWDSTART = FALSE
LDAT_ACT = LCPDAT2647
FDAT_ACT = FP2647
BAS(#CP_PARAMS, 2.0)
SET_CD_PARAMS (0)
LIN XP2647
;ENDFOLD

;FOLD LIN P2648 Vel=2 m/s CPDAT2648 Tool[1]:marker Base[0] ;%{PE}
;FOLD Parameters ;%{h}
;Params IlfProvider=kukaroboter.basistech.inlineforms.movement.old; Kuka.IsGlobalPoint=False; Kuka.PointName=P2648; Kuka.BlendingEnabled=False; Kuka.MoveDataName=CPDAT1; Kuka.VelocityPath=2; Kuka.CurrentCDSetIndex=0; Kuka.MovementParameterFieldEnabled=True; IlfCommand=LIN
;ENDFOLD
$BWDSTART = FALSE
LDAT_ACT = LCPDAT2648
FDAT_ACT = FP2648
BAS(#CP_PARAMS, 2.0)
SET_CD_PARAMS (0)
LIN XP2648
;ENDFOLD

;FOLD LIN P2649 Vel=2 m/s CPDAT2649 Tool[1]:marker Base[0] ;%{PE}
;FOLD Parameters ;%{h}
;Params IlfProvider=kukaroboter.basistech.inlineforms.movement.old; Kuka.IsGlobalPoint=False; Kuka.PointName=P2649; Kuka.BlendingEnabled=False; Kuka.MoveDataName=CPDAT1; Kuka.VelocityPath=2; Kuka.CurrentCDSetIndex=0; Kuka.MovementParameterFieldEnabled=True; IlfCommand=LIN
;ENDFOLD
$BWDSTART = FALSE
LDAT_ACT = LCPDAT2649
FDAT_ACT = FP2649
BAS(#CP_PARAMS, 2.0)
SET_CD_PARAMS (0)
LIN XP2649
;ENDFOLD

;FOLD LIN P2650 Vel=2 m/s CPDAT2650 Tool[1]:marker Base[0] ;%{PE}
;FOLD Parameters ;%{h}
;Params IlfProvider=kukaroboter.basistech.inlineforms.movement.old; Kuka.IsGlobalPoint=False; Kuka.PointName=P2650; Kuka.BlendingEnabled=False; Kuka.MoveDataName=CPDAT1; Kuka.VelocityPath=2; Kuka.CurrentCDSetIndex=0; Kuka.MovementParameterFieldEnabled=True; IlfCommand=LIN
;ENDFOLD
$BWDSTART = FALSE
LDAT_ACT = LCPDAT2650
FDAT_ACT = FP2650
BAS(#CP_PARAMS, 2.0)
SET_CD_PARAMS (0)
LIN XP2650
;ENDFOLD

;FOLD LIN P2651 Vel=2 m/s CPDAT2651 Tool[1]:marker Base[0] ;%{PE}
;FOLD Parameters ;%{h}
;Params IlfProvider=kukaroboter.basistech.inlineforms.movement.old; Kuka.IsGlobalPoint=False; Kuka.PointName=P2651; Kuka.BlendingEnabled=False; Kuka.MoveDataName=CPDAT1; Kuka.VelocityPath=2; Kuka.CurrentCDSetIndex=0; Kuka.MovementParameterFieldEnabled=True; IlfCommand=LIN
;ENDFOLD
$BWDSTART = FALSE
LDAT_ACT = LCPDAT2651
FDAT_ACT = FP2651
BAS(#CP_PARAMS, 2.0)
SET_CD_PARAMS (0)
LIN XP2651
;ENDFOLD

;FOLD LIN P2652 Vel=2 m/s CPDAT2652 Tool[1]:marker Base[0] ;%{PE}
;FOLD Parameters ;%{h}
;Params IlfProvider=kukaroboter.basistech.inlineforms.movement.old; Kuka.IsGlobalPoint=False; Kuka.PointName=P2652; Kuka.BlendingEnabled=False; Kuka.MoveDataName=CPDAT1; Kuka.VelocityPath=2; Kuka.CurrentCDSetIndex=0; Kuka.MovementParameterFieldEnabled=True; IlfCommand=LIN
;ENDFOLD
$BWDSTART = FALSE
LDAT_ACT = LCPDAT2652
FDAT_ACT = FP2652
BAS(#CP_PARAMS, 2.0)
SET_CD_PARAMS (0)
LIN XP2652
;ENDFOLD

;FOLD LIN P2653 Vel=2 m/s CPDAT2653 Tool[1]:marker Base[0] ;%{PE}
;FOLD Parameters ;%{h}
;Params IlfProvider=kukaroboter.basistech.inlineforms.movement.old; Kuka.IsGlobalPoint=False; Kuka.PointName=P2653; Kuka.BlendingEnabled=False; Kuka.MoveDataName=CPDAT1; Kuka.VelocityPath=2; Kuka.CurrentCDSetIndex=0; Kuka.MovementParameterFieldEnabled=True; IlfCommand=LIN
;ENDFOLD
$BWDSTART = FALSE
LDAT_ACT = LCPDAT2653
FDAT_ACT = FP2653
BAS(#CP_PARAMS, 2.0)
SET_CD_PARAMS (0)
LIN XP2653
;ENDFOLD

;FOLD LIN P2654 Vel=2 m/s CPDAT2654 Tool[1]:marker Base[0] ;%{PE}
;FOLD Parameters ;%{h}
;Params IlfProvider=kukaroboter.basistech.inlineforms.movement.old; Kuka.IsGlobalPoint=False; Kuka.PointName=P2654; Kuka.BlendingEnabled=False; Kuka.MoveDataName=CPDAT1; Kuka.VelocityPath=2; Kuka.CurrentCDSetIndex=0; Kuka.MovementParameterFieldEnabled=True; IlfCommand=LIN
;ENDFOLD
$BWDSTART = FALSE
LDAT_ACT = LCPDAT2654
FDAT_ACT = FP2654
BAS(#CP_PARAMS, 2.0)
SET_CD_PARAMS (0)
LIN XP2654
;ENDFOLD

;FOLD LIN P2655 Vel=2 m/s CPDAT2655 Tool[1]:marker Base[0] ;%{PE}
;FOLD Parameters ;%{h}
;Params IlfProvider=kukaroboter.basistech.inlineforms.movement.old; Kuka.IsGlobalPoint=False; Kuka.PointName=P2655; Kuka.BlendingEnabled=False; Kuka.MoveDataName=CPDAT1; Kuka.VelocityPath=2; Kuka.CurrentCDSetIndex=0; Kuka.MovementParameterFieldEnabled=True; IlfCommand=LIN
;ENDFOLD
$BWDSTART = FALSE
LDAT_ACT = LCPDAT2655
FDAT_ACT = FP2655
BAS(#CP_PARAMS, 2.0)
SET_CD_PARAMS (0)
LIN XP2655
;ENDFOLD

;FOLD LIN P2656 Vel=2 m/s CPDAT2656 Tool[1]:marker Base[0] ;%{PE}
;FOLD Parameters ;%{h}
;Params IlfProvider=kukaroboter.basistech.inlineforms.movement.old; Kuka.IsGlobalPoint=False; Kuka.PointName=P2656; Kuka.BlendingEnabled=False; Kuka.MoveDataName=CPDAT1; Kuka.VelocityPath=2; Kuka.CurrentCDSetIndex=0; Kuka.MovementParameterFieldEnabled=True; IlfCommand=LIN
;ENDFOLD
$BWDSTART = FALSE
LDAT_ACT = LCPDAT2656
FDAT_ACT = FP2656
BAS(#CP_PARAMS, 2.0)
SET_CD_PARAMS (0)
LIN XP2656
;ENDFOLD

;FOLD LIN P2657 Vel=2 m/s CPDAT2657 Tool[1]:marker Base[0] ;%{PE}
;FOLD Parameters ;%{h}
;Params IlfProvider=kukaroboter.basistech.inlineforms.movement.old; Kuka.IsGlobalPoint=False; Kuka.PointName=P2657; Kuka.BlendingEnabled=False; Kuka.MoveDataName=CPDAT1; Kuka.VelocityPath=2; Kuka.CurrentCDSetIndex=0; Kuka.MovementParameterFieldEnabled=True; IlfCommand=LIN
;ENDFOLD
$BWDSTART = FALSE
LDAT_ACT = LCPDAT2657
FDAT_ACT = FP2657
BAS(#CP_PARAMS, 2.0)
SET_CD_PARAMS (0)
LIN XP2657
;ENDFOLD

;FOLD LIN P2658 Vel=2 m/s CPDAT2658 Tool[1]:marker Base[0] ;%{PE}
;FOLD Parameters ;%{h}
;Params IlfProvider=kukaroboter.basistech.inlineforms.movement.old; Kuka.IsGlobalPoint=False; Kuka.PointName=P2658; Kuka.BlendingEnabled=False; Kuka.MoveDataName=CPDAT1; Kuka.VelocityPath=2; Kuka.CurrentCDSetIndex=0; Kuka.MovementParameterFieldEnabled=True; IlfCommand=LIN
;ENDFOLD
$BWDSTART = FALSE
LDAT_ACT = LCPDAT2658
FDAT_ACT = FP2658
BAS(#CP_PARAMS, 2.0)
SET_CD_PARAMS (0)
LIN XP2658
;ENDFOLD

;FOLD LIN P2659 Vel=2 m/s CPDAT2659 Tool[1]:marker Base[0] ;%{PE}
;FOLD Parameters ;%{h}
;Params IlfProvider=kukaroboter.basistech.inlineforms.movement.old; Kuka.IsGlobalPoint=False; Kuka.PointName=P2659; Kuka.BlendingEnabled=False; Kuka.MoveDataName=CPDAT1; Kuka.VelocityPath=2; Kuka.CurrentCDSetIndex=0; Kuka.MovementParameterFieldEnabled=True; IlfCommand=LIN
;ENDFOLD
$BWDSTART = FALSE
LDAT_ACT = LCPDAT2659
FDAT_ACT = FP2659
BAS(#CP_PARAMS, 2.0)
SET_CD_PARAMS (0)
LIN XP2659
;ENDFOLD

;FOLD LIN P2660 Vel=2 m/s CPDAT2660 Tool[1]:marker Base[0] ;%{PE}
;FOLD Parameters ;%{h}
;Params IlfProvider=kukaroboter.basistech.inlineforms.movement.old; Kuka.IsGlobalPoint=False; Kuka.PointName=P2660; Kuka.BlendingEnabled=False; Kuka.MoveDataName=CPDAT1; Kuka.VelocityPath=2; Kuka.CurrentCDSetIndex=0; Kuka.MovementParameterFieldEnabled=True; IlfCommand=LIN
;ENDFOLD
$BWDSTART = FALSE
LDAT_ACT = LCPDAT2660
FDAT_ACT = FP2660
BAS(#CP_PARAMS, 2.0)
SET_CD_PARAMS (0)
LIN XP2660
;ENDFOLD

;FOLD LIN P2661 Vel=2 m/s CPDAT2661 Tool[1]:marker Base[0] ;%{PE}
;FOLD Parameters ;%{h}
;Params IlfProvider=kukaroboter.basistech.inlineforms.movement.old; Kuka.IsGlobalPoint=False; Kuka.PointName=P2661; Kuka.BlendingEnabled=False; Kuka.MoveDataName=CPDAT1; Kuka.VelocityPath=2; Kuka.CurrentCDSetIndex=0; Kuka.MovementParameterFieldEnabled=True; IlfCommand=LIN
;ENDFOLD
$BWDSTART = FALSE
LDAT_ACT = LCPDAT2661
FDAT_ACT = FP2661
BAS(#CP_PARAMS, 2.0)
SET_CD_PARAMS (0)
LIN XP2661
;ENDFOLD

;FOLD LIN P2662 Vel=2 m/s CPDAT2662 Tool[1]:marker Base[0] ;%{PE}
;FOLD Parameters ;%{h}
;Params IlfProvider=kukaroboter.basistech.inlineforms.movement.old; Kuka.IsGlobalPoint=False; Kuka.PointName=P2662; Kuka.BlendingEnabled=False; Kuka.MoveDataName=CPDAT1; Kuka.VelocityPath=2; Kuka.CurrentCDSetIndex=0; Kuka.MovementParameterFieldEnabled=True; IlfCommand=LIN
;ENDFOLD
$BWDSTART = FALSE
LDAT_ACT = LCPDAT2662
FDAT_ACT = FP2662
BAS(#CP_PARAMS, 2.0)
SET_CD_PARAMS (0)
LIN XP2662
;ENDFOLD

;FOLD LIN P2663 Vel=2 m/s CPDAT2663 Tool[1]:marker Base[0] ;%{PE}
;FOLD Parameters ;%{h}
;Params IlfProvider=kukaroboter.basistech.inlineforms.movement.old; Kuka.IsGlobalPoint=False; Kuka.PointName=P2663; Kuka.BlendingEnabled=False; Kuka.MoveDataName=CPDAT1; Kuka.VelocityPath=2; Kuka.CurrentCDSetIndex=0; Kuka.MovementParameterFieldEnabled=True; IlfCommand=LIN
;ENDFOLD
$BWDSTART = FALSE
LDAT_ACT = LCPDAT2663
FDAT_ACT = FP2663
BAS(#CP_PARAMS, 2.0)
SET_CD_PARAMS (0)
LIN XP2663
;ENDFOLD

;FOLD LIN P2664 Vel=2 m/s CPDAT2664 Tool[1]:marker Base[0] ;%{PE}
;FOLD Parameters ;%{h}
;Params IlfProvider=kukaroboter.basistech.inlineforms.movement.old; Kuka.IsGlobalPoint=False; Kuka.PointName=P2664; Kuka.BlendingEnabled=False; Kuka.MoveDataName=CPDAT1; Kuka.VelocityPath=2; Kuka.CurrentCDSetIndex=0; Kuka.MovementParameterFieldEnabled=True; IlfCommand=LIN
;ENDFOLD
$BWDSTART = FALSE
LDAT_ACT = LCPDAT2664
FDAT_ACT = FP2664
BAS(#CP_PARAMS, 2.0)
SET_CD_PARAMS (0)
LIN XP2664
;ENDFOLD

